REGION Network 26: pomocniczy bit ustawiania pompy dodatkowej nr1
   // Reset znacznika po udanym załączeniu pompy dodatkowej
   // Reset w wypadku braku pompy
   RUNG wire#powerrail
      I_Contact( "AlwaysTRUE" )
      wire#w1
      Contact( "Is_extras_K1_P1" )
      Contact( "IsRunNetwork_P1" )
      wire#w2
      R_Coil( #set_Motor2 )
   END_RUNG
   RUNG wire#w1
      Contact( "Is_extras_K1_P2" )
      Contact( "IsRunNetwork_P2" )
   END_RUNG wire#w2
   RUNG wire#w1
      Contact( "Is_extras_K1_P3" )
      Contact( "IsRunNetwork_P3" )
   END_RUNG wire#w2
   RUNG wire#w1
      Contact( "Is_extras_K1_P4" )
      Contact( "IsRunNetwork_P4" )
   END_RUNG wire#w2
   RUNG wire#w1
      Contact( "Reset_Motor2Alarm" )
   END_RUNG wire#w2
   RUNG wire#w1
      I_Contact( "IsModeAut" )
   END_RUNG wire#w2
   // the same network as SCL:
   IF NOT "AlwaysTRUE" AND (("Is_extras_K1_P1" AND "IsRunNetwork_P1") OR ("Is_extras_K1_P2" AND "IsRunNetwork_P2") OR ("Is_extras_K1_P3" AND "IsRunNetwork_P3") OR ("Is_extras_K1_P4" AND "IsRunNetwork_P4") OR "Reset_Motor2Alarm" OR NOT "IsModeAut") THEN
       #set_Motor2 := FALSE;
   END_IF;
END_REGION

REGION Network 27: pomocniczy bit ustawiania pompy dodatkoweo nr2
   // Reset znacznika po udanym załączeniu pompy dodatkowej
   // Reset w wypadku braku pompy
   RUNG wire#powerrail
      I_Contact( "AlwaysTRUE" )
      wire#w1
      Contact( "Is_extras_K2_P1" )
      Contact( "IsRunNetwork_P1" )
      wire#w2
      R_Coil( #set_Motor3 )
   END_RUNG
   RUNG wire#w1
      Contact( "Is_extras_K2_P2" )
      Contact( "IsRunNetwork_P2" )
   END_RUNG wire#w2
   RUNG wire#w1
      Contact( "Is_extras_K2_P3" )
      Contact( "IsRunNetwork_P3" )
   END_RUNG wire#w2
   RUNG wire#w1
      Contact( "Is_extras_K2_P4" )
      Contact( "IsRunNetwork_P4" )
   END_RUNG wire#w2
   RUNG wire#w1
      Contact( "Reset_Motor3Alarm" )
   END_RUNG wire#w2
   RUNG wire#w1
      I_Contact( "IsModeAut" )
   END_RUNG wire#w2
   // the same network as SCL:
   IF NOT "AlwaysTRUE" AND (("Is_extras_K2_P1" AND "IsRunNetwork_P1") OR ("Is_extras_K2_P2" AND "IsRunNetwork_P2") OR ("Is_extras_K2_P3" AND "IsRunNetwork_P3") OR ("Is_extras_K2_P4" AND "IsRunNetwork_P4") OR "Reset_Motor3Alarm" OR NOT "IsModeAut") THEN
       #set_Motor3 := FALSE;
   END_IF;
END_REGION

REGION Network 28: pomocniczy bit ustawiania pompy dodatkowe nr3
   // Reset znacznika po udanym załączeniu pompy dodatkowej
   // Reset w wypadku braku pompy
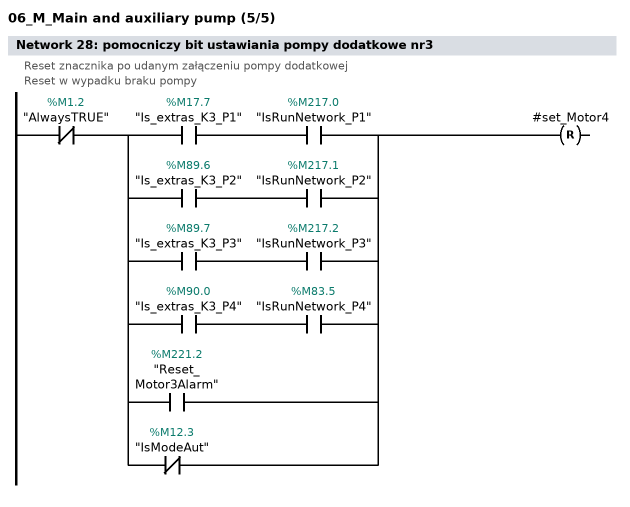
   RUNG wire#powerrail
      I_Contact( "AlwaysTRUE" )
      wire#w1
      Contact( "Is_extras_K3_P1" )
      Contact( "IsRunNetwork_P1" )
      wire#w2
      R_Coil( #set_Motor4 )
   END_RUNG
   RUNG wire#w1
      Contact( "Is_extras_K3_P2" )
      Contact( "IsRunNetwork_P2" )
   END_RUNG wire#w2
   RUNG wire#w1
      Contact( "Is_extras_K3_P3" )
      Contact( "IsRunNetwork_P3" )
   END_RUNG wire#w2
   RUNG wire#w1
      Contact( "Is_extras_K3_P4" )
      Contact( "IsRunNetwork_P4" )
   END_RUNG wire#w2
   RUNG wire#w1
      Contact( "Reset_Motor3Alarm" )
   END_RUNG wire#w2
   RUNG wire#w1
      I_Contact( "IsModeAut" )
   END_RUNG wire#w2
   // the same network as SCL:
   IF NOT "AlwaysTRUE" AND (("Is_extras_K3_P1" AND "IsRunNetwork_P1") OR ("Is_extras_K3_P2" AND "IsRunNetwork_P2") OR ("Is_extras_K3_P3" AND "IsRunNetwork_P3") OR ("Is_extras_K3_P4" AND "IsRunNetwork_P4") OR "Reset_Motor3Alarm" OR NOT "IsModeAut") THEN
       #set_Motor4 := FALSE;
   END_IF;
END_REGION
END_FUNCTION_BLOCK

FUNCTION_BLOCK "06_M_Inverter connection control"   // FB8, LAD
TITLE = Sterowanie dołączaniem styczników falownika
{ S7_Optimized_Access := 'TRUE' }
AUTHOR : rtecmer
VERSION : 0.1
// Sterowa stycznikiem pracy z falownika.
// Funkcja FB8 komutuje załaczenie stycznika FALOWNIK dla konkretnego napędu. Napędem sterowanym jest zawsze napęd przypisany do MC (czyli IsReady_MC to jest gotowość napędu sterowaniego) Na wejścia oznaczone wyróżnikiem MC podlączamy sygnały tej samej dmuchawy, której stycznikiem będziemy sterować poprzez wtjście setSUPV_FM
//  
// Sterowanie stycznikiem . Ustawianie znaczników setCMD_FM i setSUPV_FM które przekazywane są do funkcji FC3/FC1 DRV01 driver napędów. Następnie przekazywane jest do warstwy Hawtware/ OUT gdzie ustawiane jest wyjście sterownika
// stored: AutoNumber true, IsIECCheckEnabled false, IsRetainMemResEnabled false, MemoryReserve 500, SetENOAutomatically false, UDAEnableTagReadback false
   VAR_INPUT
      Is_up_Hz : Bool;
      Set_HWork_M : Bool;   // Znacznik ustawienia pracy od licznika
      setPID_Pompy : Bool;   // Znacznik załączenie, regulacji falownika
      IsRunInverter_MA : Bool;   // Potwierdzenie pracy z falownika kompresor dodatkowy 1
      IsRunNetwork_MA : Bool;   // Potwierdzenie praca z sieć dodatkowego
      IsRunInverter_MB : Bool;   // Potwierdzenie pracy z falownika kompresor dodatkowy 2
      IsRunNetwork_MB : Bool;   // Potwierdzenie praca z sieć dodatkowego
      IsRunNetwork_MC : Bool;   // Potwierdzenie pracy z sieci
      IsRunInverter_MC : Bool;   // Potwierdzenie pracy z falownika
      IsRunNetwork_MD : Bool;   // Potwierdzenie pracy z sieci
      IsRunInverter_MD : Bool;   // Potwierdzenie pracy z falownika
      FC2_Set_50H : Bool;   // Znacznik osiągnięcia czasu dla 50Hz
      IsRunInverter1 : Bool;   // Potwierdzenie pracy falownika
      AlwaysTRUE : Bool;
      IsReady_MA : Bool;   // Znacznik gotowości
      IsReady_MB : Bool;   // Znacznik gotowości
      IsReady_MC : Bool;   // Znacznik gotowości
      IsReady_MD : Bool;   // Znacznik gotowości
      IsModeAut : Bool;   // Znacznik trybu automat
      FB9_Set_Motor2 : Bool;   // Polecenie dostawienia dodatkowej nr1
      FB9_Set_Motor3 : Bool;   // Polecenie dostawienia dodatkowej nr2
      FB9_Set_Motor4 : Bool;   // Polecenie dostawienia dodatkowej nr3
      IsReady_Inverter : Bool;   // Gotowość falownika
      ResWorkInverter_to_MaxTime : Bool;   // Bit kasowania pracy falownika od maxymalnej ciągłej pracy
      number_pump : Int;   // numer pompy w instalacji
      ActivePump : Int;   // numer pompy wiodącej
   END_VAR
   VAR_OUTPUT
      setSUPV_FM : Bool;   // Znacznik polecenia startu z falownika
   END_VAR
   VAR_IN_OUT
      setCMD_FM : Bool;   // Znacznik sterowania w trybie falownik
      Timer_OFF_Inverter_M : TOF_TIME;   // Timer na blokowanie po odłączeniu stycznika falownika
      Timer_Start_Inver_M : TON_TIME;   // Timer opóźnienia załaczenia stycznika pracy z falownika
      Timer_Set50Hz_Off_Inver_M : TON_TIME;   // Timer opóźnieniawyłączeniea falownika
      Mem_Res_setCMD_MC : Bool;   // pamięć zbocza załączenia timera blokowania stycznika falowni
   END_VAR
   VAR
      IsDrive_Optimum { ExternalAccessible := 'False'; ExternalVisible := 'False'; ExternalWritable := 'False'} : Bool;   // Znacznik optymalnej ilości napędów. Jeśli False to nie przełaczaj Falowni/Sieć
      CMD_OFF_inverter { ExternalAccessible := 'False'; ExternalVisible := 'False'; ExternalWritable := 'False'} : Bool;   // Wyłączenie falownika od 50Hz i dodatkowa
      tmpOFF_inverter { ExternalAccessible := 'False'; ExternalVisible := 'False'; ExternalWritable := 'False'} : Bool;
      Network_50Hz : Bool;   // Znacznik 50 Hz podtrzymanie przełączenia na sieć
   END_VAR
   VAR_TEMP   // added for the SCL form of the ladder/FBD networks
      _w1 : Bool;
      _w2 : Bool;
   END_VAR
BEGIN

REGION Network 1: Kontrola statusu napędu
END_REGION

REGION Network 2: Histereza na dołączenie stycznika falownika
   // Sterowanie dołączeniem stycznika pracy z falownika
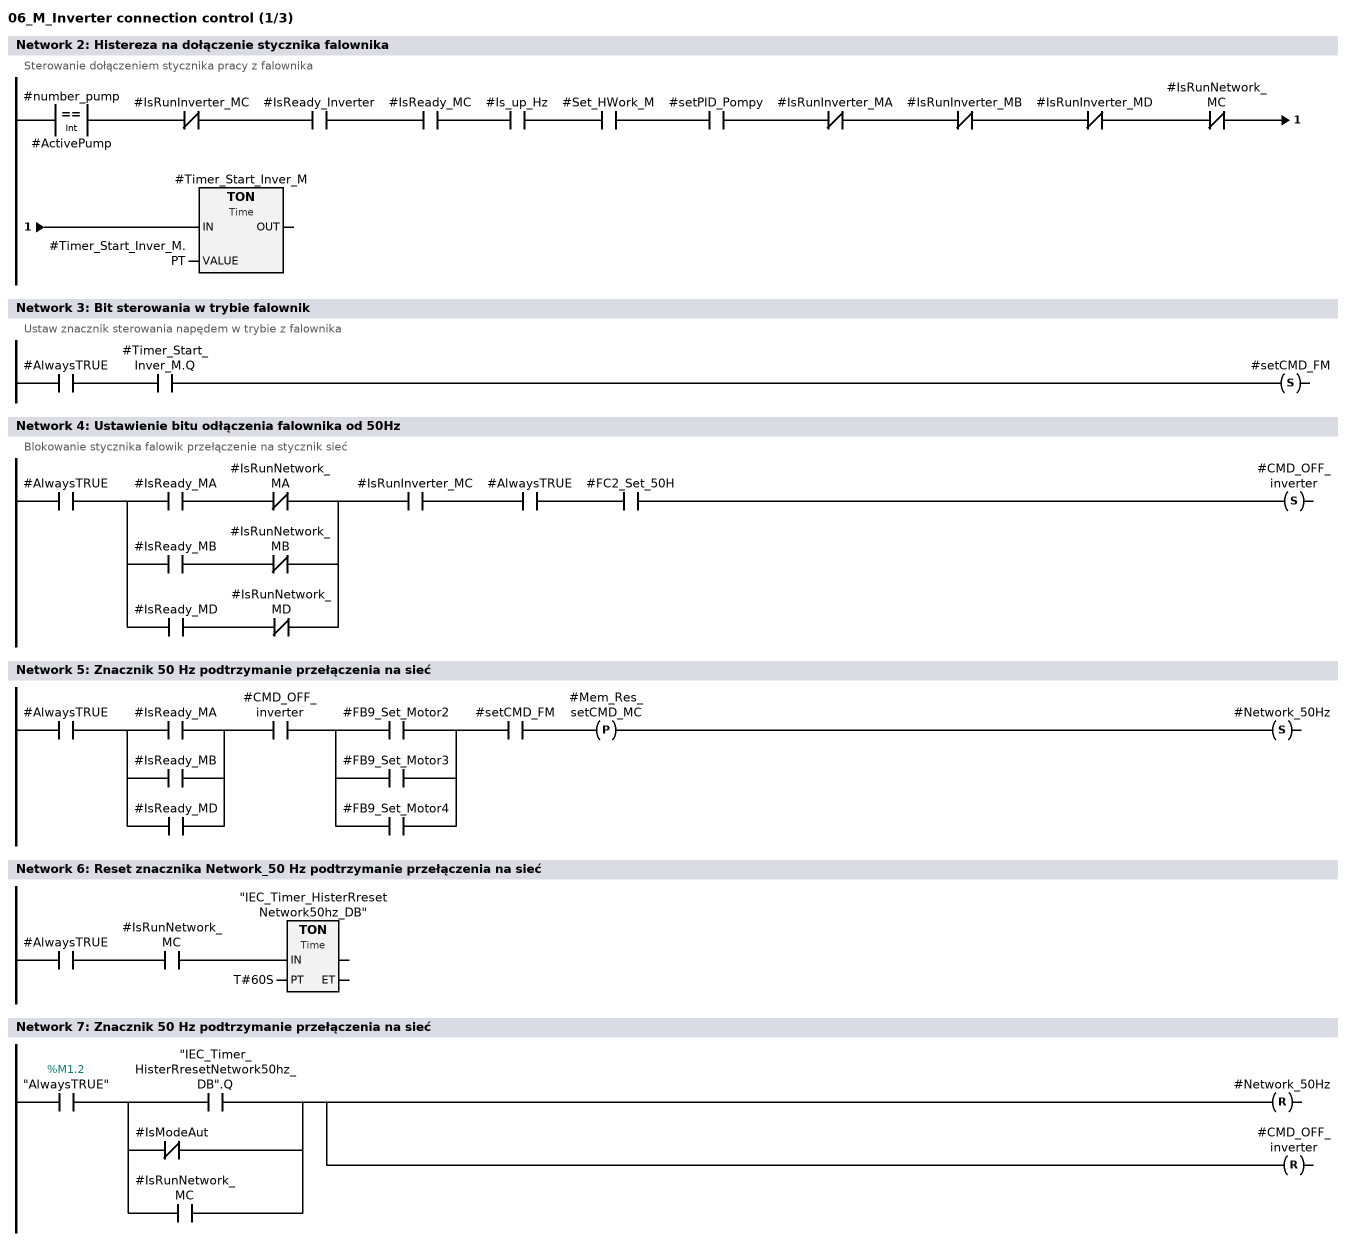
   #Timer_Start_Inver_M(IN := (#number_pump = #ActivePump) AND NOT #IsRunInverter_MC AND #IsReady_Inverter AND #IsReady_MC AND #Is_up_Hz AND #Set_HWork_M AND #setPID_Pompy AND NOT #IsRunInverter_MA AND NOT #IsRunInverter_MB AND NOT #IsRunInverter_MD AND NOT #IsRunNetwork_MC, PT := #Timer_Start_Inver_M.PT);   // TON coil
END_REGION

REGION Network 3: Bit sterowania w trybie falownik
   // Ustaw znacznik sterowania napędem w trybie z falownika
   RUNG wire#powerrail
      Contact( #AlwaysTRUE )
      Contact( #Timer_Start_Inver_M.Q )
      S_Coil( #setCMD_FM )
   END_RUNG
   // the same network as SCL:
   IF #AlwaysTRUE AND #Timer_Start_Inver_M.Q THEN #setCMD_FM := TRUE; END_IF;
END_REGION

REGION Network 4: Ustawienie bitu odłączenia falownika od 50Hz
   // Blokowanie stycznika falowik przełączenie na stycznik sieć
   RUNG wire#powerrail
      Contact( #AlwaysTRUE )
      wire#w1
      Contact( #IsReady_MA )
      I_Contact( #IsRunNetwork_MA )
      wire#w2
      Contact( #IsRunInverter_MC )
      Contact( #AlwaysTRUE )
      Contact( #FC2_Set_50H )
      S_Coil( #CMD_OFF_inverter )
   END_RUNG
   RUNG wire#w1
      Contact( #IsReady_MB )
      I_Contact( #IsRunNetwork_MB )
   END_RUNG wire#w2
   RUNG wire#w1
      Contact( #IsReady_MD )
      I_Contact( #IsRunNetwork_MD )
   END_RUNG wire#w2
   // the same network as SCL:
   IF #AlwaysTRUE AND ((#IsReady_MA AND NOT #IsRunNetwork_MA) OR (#IsReady_MB AND NOT #IsRunNetwork_MB) OR (#IsReady_MD AND NOT #IsRunNetwork_MD)) AND #IsRunInverter_MC AND #AlwaysTRUE AND #FC2_Set_50H THEN
       #CMD_OFF_inverter := TRUE;
   END_IF;
END_REGION

REGION Network 5: Znacznik 50 Hz podtrzymanie przełączenia na sieć
   RUNG wire#powerrail
      Contact( #AlwaysTRUE )
      wire#w1
      Contact( #IsReady_MA )
      wire#w2
      Contact( #CMD_OFF_inverter )
      wire#w3
      Contact( #FB9_Set_Motor2 )
      wire#w4
      Contact( #setCMD_FM )
      P_Trig( #Mem_Res_setCMD_MC )
      S_Coil( #Network_50Hz )
   END_RUNG
   RUNG wire#w1
      Contact( #IsReady_MB )
   END_RUNG wire#w2
   RUNG wire#w1
      Contact( #IsReady_MD )
   END_RUNG wire#w2
   RUNG wire#w3
      Contact( #FB9_Set_Motor3 )
   END_RUNG wire#w4
   RUNG wire#w3
      Contact( #FB9_Set_Motor4 )
   END_RUNG wire#w4
   // the same network as SCL:
   #_w1 := #AlwaysTRUE AND (#IsReady_MA OR #IsReady_MB OR #IsReady_MD) AND #CMD_OFF_inverter AND (#FB9_Set_Motor2 OR #FB9_Set_Motor3 OR #FB9_Set_Motor4) AND #setCMD_FM;
   #_w2 := #_w1 AND NOT #Mem_Res_setCMD_MC;   // rising edge
   #Mem_Res_setCMD_MC := #_w1;
   IF #_w2 THEN #Network_50Hz := TRUE; END_IF;
END_REGION

REGION Network 6: Reset znacznika Network_50 Hz podtrzymanie przełączenia na sieć
   RUNG wire#powerrail
      Contact( #AlwaysTRUE )
      Contact( #IsRunNetwork_MC )
      { S7_Templates := "time_type := Time" } "IEC_Timer_HisterRresetNetwork50hz_DB".TON(pt := T#60S, et =>)
   END_RUNG
   // the same network as SCL:
   "IEC_Timer_HisterRresetNetwork50hz_DB".TON(IN := #AlwaysTRUE AND #IsRunNetwork_MC, PT := T#60S);
END_REGION

REGION Network 7: Znacznik 50 Hz podtrzymanie przełączenia na sieć
   RUNG wire#powerrail
      Contact( "AlwaysTRUE" )
      wire#w1
      Contact( "IEC_Timer_HisterRresetNetwork50hz_DB".Q )
      wire#w2
      R_Coil( #Network_50Hz )
   END_RUNG
   RUNG wire#w1
      I_Contact( #IsModeAut )
   END_RUNG wire#w2
   RUNG wire#w1
      Contact( #IsRunNetwork_MC )
   END_RUNG wire#w2
   RUNG wire#w2
      R_Coil( #CMD_OFF_inverter )
   END_RUNG
   // the same network as SCL:
   IF "AlwaysTRUE" AND ("IEC_Timer_HisterRresetNetwork50hz_DB".Q OR NOT #IsModeAut OR #IsRunNetwork_MC) THEN
       #Network_50Hz := FALSE;
       #CMD_OFF_inverter := FALSE;
   END_IF;
END_REGION

REGION Network 8: Timer blokowania po odłączenieu stycznika falownik
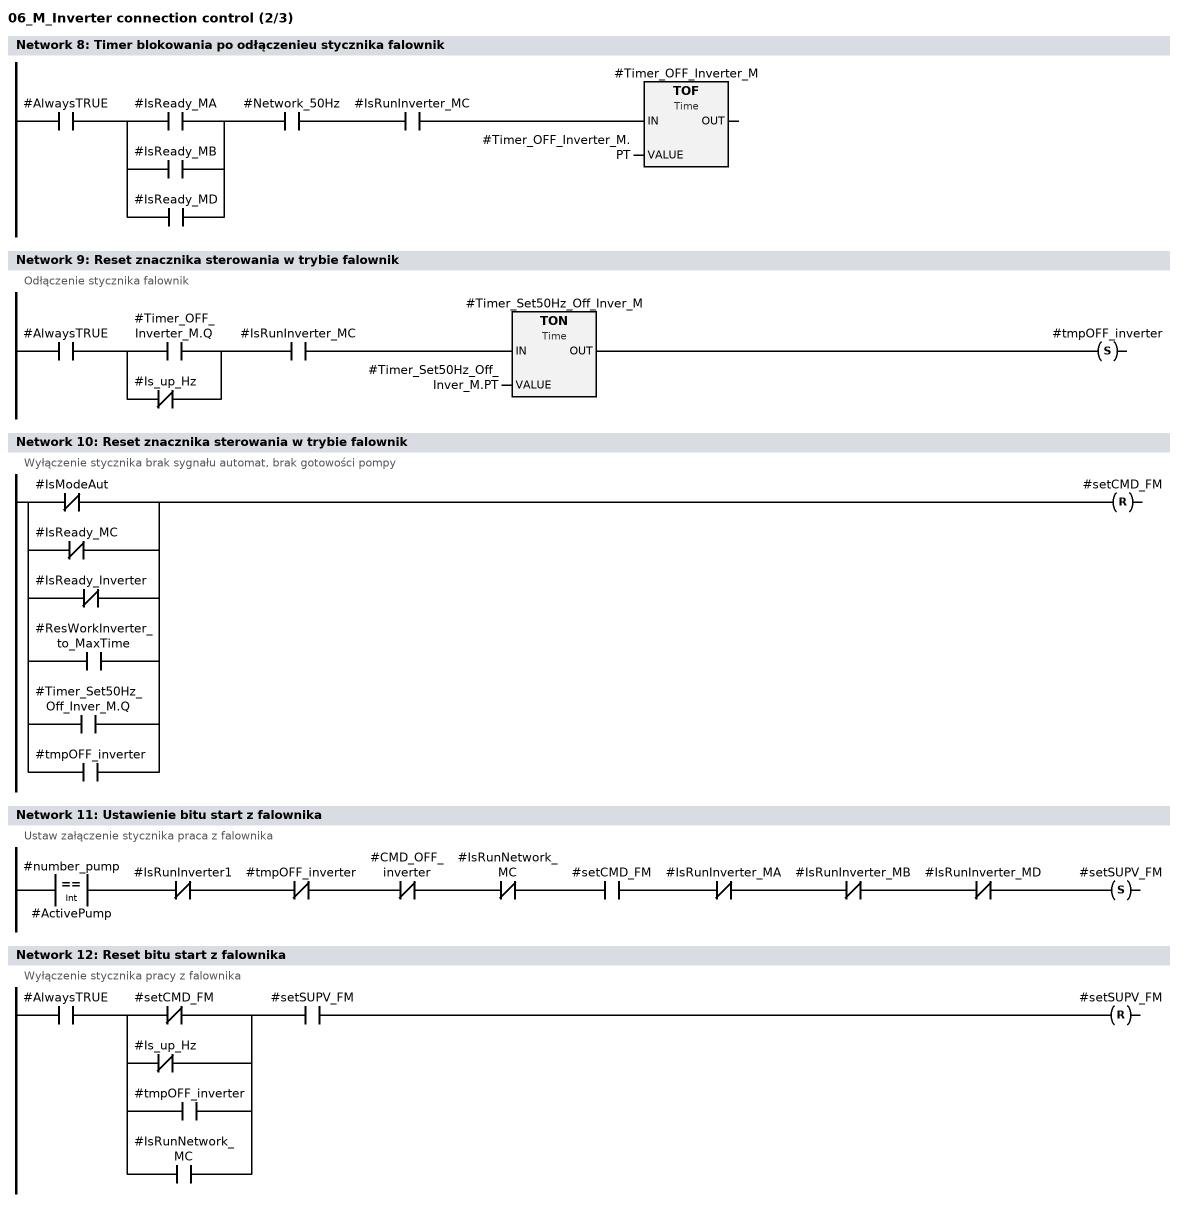
   #Timer_OFF_Inverter_M(IN := #AlwaysTRUE AND (#IsReady_MA OR #IsReady_MB OR #IsReady_MD) AND #Network_50Hz AND #IsRunInverter_MC, PT := #Timer_OFF_Inverter_M.PT);   // TOF coil
END_REGION

REGION Network 9: Reset znacznika sterowania w trybie falownik
   // Odłączenie stycznika falownik
   #_w1 := #AlwaysTRUE AND (#Timer_OFF_Inverter_M.Q OR NOT #Is_up_Hz) AND #IsRunInverter_MC;
   #Timer_Set50Hz_Off_Inver_M(IN := #_w1, PT := #Timer_Set50Hz_Off_Inver_M.PT);   // TON coil
   IF #_w1 THEN #tmpOFF_inverter := TRUE; END_IF;
END_REGION

REGION Network 10: Reset znacznika sterowania w trybie falownik
   // Wyłączenie stycznika brak sygnału automat, brak gotowości pompy
   RUNG wire#powerrail
      I_Contact( #IsModeAut )
      wire#w1
      R_Coil( #setCMD_FM )
   END_RUNG
   RUNG wire#powerrail
      I_Contact( #IsReady_MC )
   END_RUNG wire#w1
   RUNG wire#powerrail
      I_Contact( #IsReady_Inverter )
   END_RUNG wire#w1
   RUNG wire#powerrail
      Contact( #ResWorkInverter_to_MaxTime )
   END_RUNG wire#w1
   RUNG wire#powerrail
      Contact( #Timer_Set50Hz_Off_Inver_M.Q )
   END_RUNG wire#w1
   RUNG wire#powerrail
      Contact( #tmpOFF_inverter )
   END_RUNG wire#w1
   // the same network as SCL:
   IF NOT #IsModeAut OR NOT #IsReady_MC OR NOT #IsReady_Inverter OR #ResWorkInverter_to_MaxTime OR #Timer_Set50Hz_Off_Inver_M.Q OR #tmpOFF_inverter THEN
       #setCMD_FM := FALSE;
   END_IF;
END_REGION

REGION Network 11: Ustawienie bitu start z falownika
   // Ustaw załączenie stycznika praca z falownika
   RUNG wire#powerrail
      { S7_Templates := "SrcType := Int" } EQ_Contact(in1 := #number_pump, in2 := #ActivePump)
      I_Contact( #IsRunInverter1 )
      I_Contact( #tmpOFF_inverter )
      I_Contact( #CMD_OFF_inverter )
      I_Contact( #IsRunNetwork_MC )
      Contact( #setCMD_FM )
      I_Contact( #IsRunInverter_MA )
      I_Contact( #IsRunInverter_MB )
      I_Contact( #IsRunInverter_MD )
      S_Coil( #setSUPV_FM )
   END_RUNG
   // the same network as SCL:
   IF (#number_pump = #ActivePump) AND NOT #IsRunInverter1 AND NOT #tmpOFF_inverter AND NOT #CMD_OFF_inverter AND NOT #IsRunNetwork_MC AND #setCMD_FM AND NOT #IsRunInverter_MA AND NOT #IsRunInverter_MB AND NOT #IsRunInverter_MD THEN
       #setSUPV_FM := TRUE;
   END_IF;
END_REGION

REGION Network 12: Reset bitu start z falownika
   // Wyłączenie stycznika pracy z falownika
   RUNG wire#powerrail
      Contact( #AlwaysTRUE )
      wire#w1
      I_Contact( #setCMD_FM )
      wire#w2
      Contact( #setSUPV_FM )
      R_Coil( #setSUPV_FM )
   END_RUNG
   RUNG wire#w1
      I_Contact( #Is_up_Hz )
   END_RUNG wire#w2
   RUNG wire#w1
      Contact( #tmpOFF_inverter )
   END_RUNG wire#w2
   RUNG wire#w1
      Contact( #IsRunNetwork_MC )
   END_RUNG wire#w2
   // the same network as SCL:
   IF #AlwaysTRUE AND (NOT #setCMD_FM OR NOT #Is_up_Hz OR #tmpOFF_inverter OR #IsRunNetwork_MC) AND #setSUPV_FM THEN
       #setSUPV_FM := FALSE;
   END_IF;
END_REGION

REGION Network 13: Znacznik polecenia stop z falownika
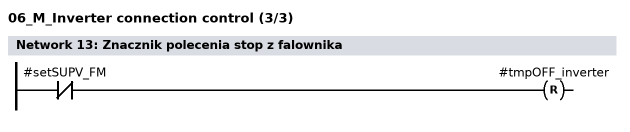
   RUNG wire#powerrail
      I_Contact( #setSUPV_FM )
      R_Coil( #tmpOFF_inverter )
   END_RUNG
   // the same network as SCL:
   IF NOT #setSUPV_FM THEN #tmpOFF_inverter := FALSE; END_IF;
END_REGION
END_FUNCTION_BLOCK

FUNCTION "06_M_Working Mode Correction" : Void   // FC34, LAD
TITLE = potrzymanie trybu
{ S7_Optimized_Access := 'TRUE' }
AUTHOR : rtecmer
VERSION : 0.1
// z powodu P1 dodanyblok potzymujący tryb pracy napędów podczas przełączania falowni / siec
// stored: AutoNumber true, IsIECCheckEnabled false, SetENOAutomatically false, UDAEnableTagReadback false
   VAR_TEMP   // added for the SCL form of the ladder/FBD networks
      _w1 : Bool;
   END_VAR
BEGIN

REGION Network 2: Ustawienie pracy [Automat]
   // Ustawienie bitu [Automat] przełacznikiem trybu pracy
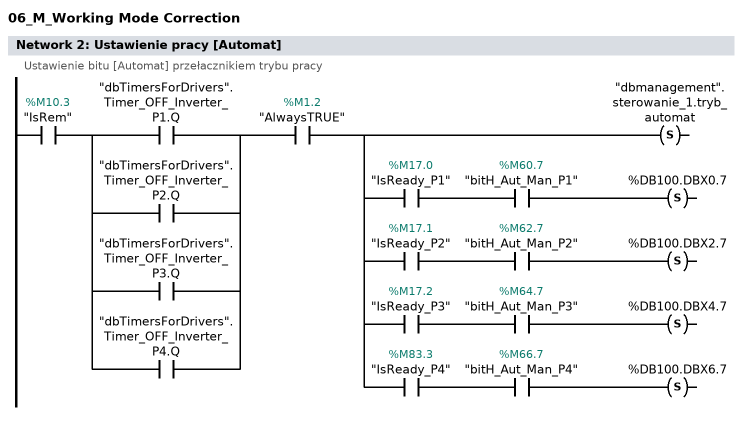
   RUNG wire#powerrail
      Contact( "IsRem" )
      wire#w1
      Contact( "dbTimersForDrivers".Timer_OFF_Inverter_P1.Q )
      wire#w2
      Contact( "AlwaysTRUE" )
      wire#w3
      S_Coil( "dbmanagement".sterowanie_1.tryb_automat )
   END_RUNG
   RUNG wire#w1
      Contact( "dbTimersForDrivers".Timer_OFF_Inverter_P2.Q )
   END_RUNG wire#w2
   RUNG wire#w1
      Contact( "dbTimersForDrivers".Timer_OFF_Inverter_P3.Q )
   END_RUNG wire#w2
   RUNG wire#w1
      Contact( "dbTimersForDrivers".Timer_OFF_Inverter_P4.Q )
   END_RUNG wire#w2
   RUNG wire#w3
      Contact( "IsReady_P1" )
      Contact( "bitH_Aut_Man_P1" )
      S_Coil( %DB100.DBX0.7 )
   END_RUNG
   RUNG wire#w3
      Contact( "IsReady_P2" )
      Contact( "bitH_Aut_Man_P2" )
      S_Coil( %DB100.DBX2.7 )
   END_RUNG
   RUNG wire#w3
      Contact( "IsReady_P3" )
      Contact( "bitH_Aut_Man_P3" )
      S_Coil( %DB100.DBX4.7 )
   END_RUNG
   RUNG wire#w3
      Contact( "IsReady_P4" )
      Contact( "bitH_Aut_Man_P4" )
      S_Coil( %DB100.DBX6.7 )
   END_RUNG
   // the same network as SCL:
   #_w1 := "IsRem" AND ("dbTimersForDrivers".Timer_OFF_Inverter_P1.Q OR "dbTimersForDrivers".Timer_OFF_Inverter_P2.Q OR "dbTimersForDrivers".Timer_OFF_Inverter_P3.Q OR "dbTimersForDrivers".Timer_OFF_Inverter_P4.Q) AND "AlwaysTRUE";
   IF #_w1 THEN "dbmanagement".sterowanie_1.tryb_automat := TRUE; END_IF;
   IF #_w1 AND "IsReady_P1" AND "bitH_Aut_Man_P1" THEN %DB100.DBX0.7 := TRUE; END_IF;
   IF #_w1 AND "IsReady_P2" AND "bitH_Aut_Man_P2" THEN %DB100.DBX2.7 := TRUE; END_IF;
   IF #_w1 AND "IsReady_P3" AND "bitH_Aut_Man_P3" THEN %DB100.DBX4.7 := TRUE; END_IF;
   IF #_w1 AND "IsReady_P4" AND "bitH_Aut_Man_P4" THEN %DB100.DBX6.7 := TRUE; END_IF;
END_REGION
END_FUNCTION

FUNCTION_BLOCK "06_M_Inverte control"   // FB11, LAD
TITLE = Control of Inverters
{ S7_Optimized_Access := 'TRUE' }
AUTHOR : rtecmer
VERSION : 0.1
// Sterowanie przekaćnikiem załączającym falownik do pracy
// stored: AutoNumber true, IsIECCheckEnabled false, IsRetainMemResEnabled false, MemoryReserve 500, SetENOAutomatically false, UDAEnableTagReadback false
   VAR_INPUT
      IsModeAut : Bool;   // Znacznik tryb automat dla pomp
      AlwaysTRUE : Bool;
      Set_HWork_P1 : Bool;   // Znacznik ustawienia pracy od licznika pracy
      Set_HWork_P2 : Bool;   // Znacznik ustawienia pracy od licznika pracy
      Set_HWork_P3 : Bool;   // Znacznik ustawienia pracy od licznika pracy
      Set_HWork_P4 : Bool;
      setPID_Pomp : Bool;   // Znacznik załączenie, regulacji falownika
      Is_loading_K3 : Bool;   // Znacznik pompy wiodącej
      IsRunInverter_P4 : Bool;
      IsRunInverter_P3 : Bool;   // Potwierdzenie załączenie stycznika falownik pompy
      IsRunInverter_P2 : Bool;   // Potwierdzenie załączenie stycznika falownik pompy
      IsRunInverter_P1 : Bool;   // Potwierdzenie załączenie stycznika falownik pompy
      Bit_Aut_P1 : Bool;   // Bit tryb prac automat
      Bit_Aut_P2 : Bool;   // Bit tryb prac automat
      Bit_Aut_P3 : Bool;   // Bit tryb prac automat
      Bit_Aut_P4 : Bool;
      IsRunNetwork_P1 : Bool;   // Potwierdzenie załączenie stycznika sieć
      IsRunNetwork_P2 : Bool := false;   // Potwierdzenie załączenie stycznika sieć
      IsRunNetwork_P3 : Bool := false;   // Potwierdzenie załączenie stycznika sieć
      IsRunNetwork_P4 : Bool;
   END_VAR
   VAR_OUTPUT
      CMD_start_stop_inverter : Bool;   // Przekaźnik sterowania załączaniem falownika
   END_VAR
   VAR
      Res_upHz : Bool;   // Reset znacznika up_Hz wyłaczenie dodatkowe
   END_VAR
BEGIN

REGION Network 1: Reset bitu pomocniczego ustalenia przyrostu Hz
   // Kasowanie podczas rozruchu po restarcie
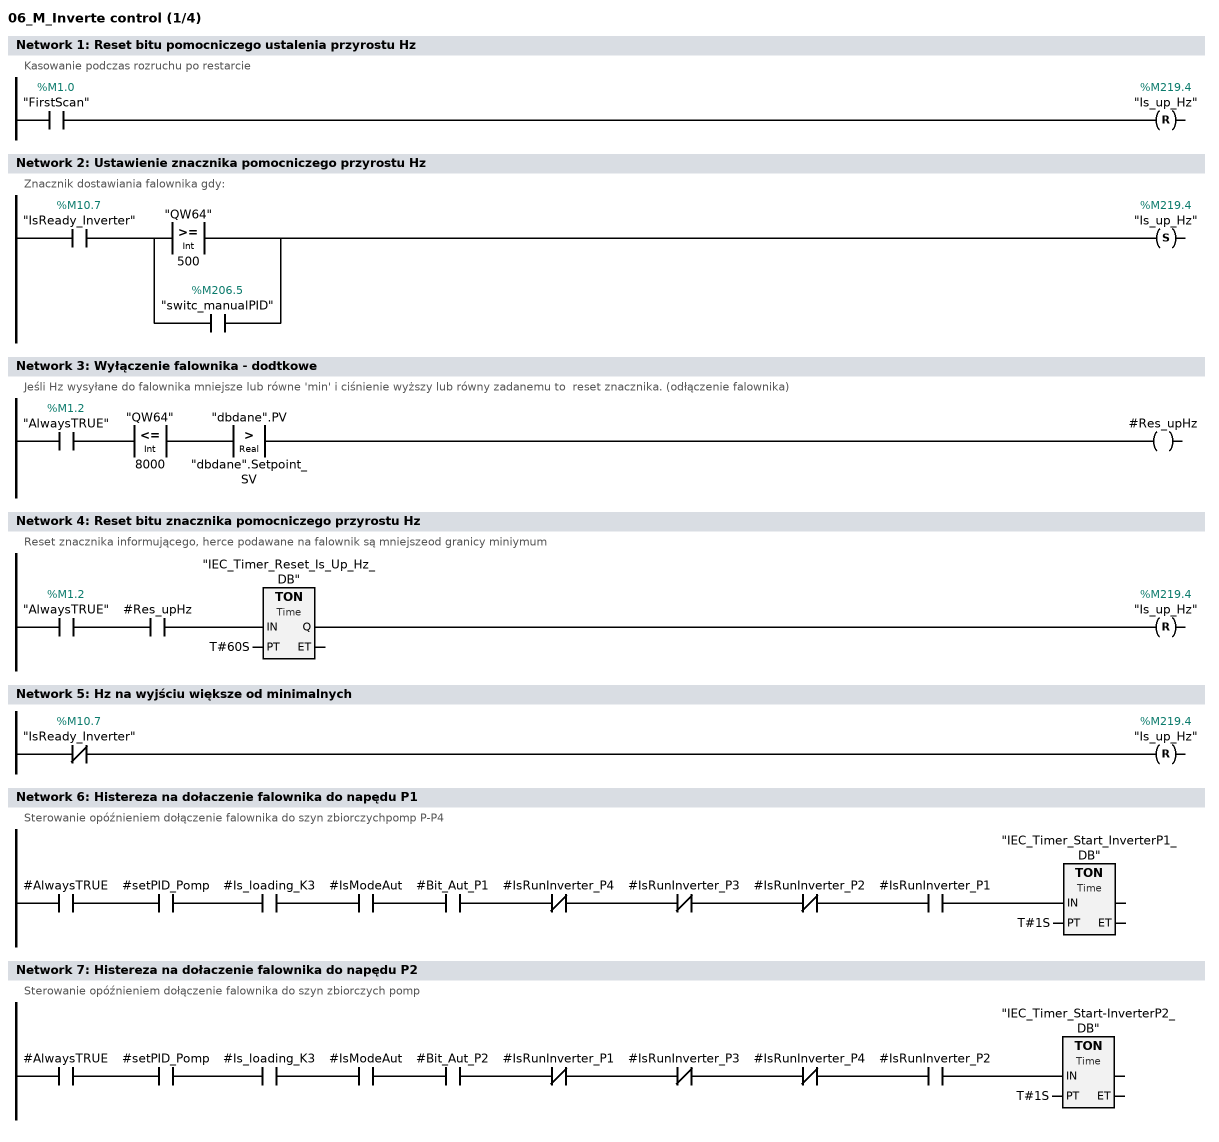
   RUNG wire#powerrail
      Contact( "FirstScan" )
      R_Coil( "Is_up_Hz" )
   END_RUNG
   // the same network as SCL:
   IF "FirstScan" THEN "Is_up_Hz" := FALSE; END_IF;
END_REGION

REGION Network 2: Ustawienie znacznika pomocniczego przyrostu Hz
   // Znacznik dostawiania falownika gdy:
   RUNG wire#powerrail
      Contact( "IsReady_Inverter" )
      wire#w1
      { S7_Templates := "SrcType := Int" } GE_Contact(in1 := "QW64", in2 := 500)
      wire#w2
      S_Coil( "Is_up_Hz" )
   END_RUNG
   RUNG wire#w1
      Contact( "switc_manualPID" )
   END_RUNG wire#w2
   // the same network as SCL:
   IF "IsReady_Inverter" AND (("QW64" >= 500) OR "switc_manualPID") THEN "Is_up_Hz" := TRUE; END_IF;
END_REGION

REGION Network 3: Wyłączenie falownika - dodtkowe
   // Jeśli Hz wysyłane do falownika mniejsze lub równe 'min' i ciśnienie wyższy lub równy zadanemu to  reset znacznika. (odłączenie falownika)
   RUNG wire#powerrail
      Contact( "AlwaysTRUE" )
      { S7_Templates := "SrcType := Int" } LE_Contact(in1 := "QW64", in2 := 8000)
      { S7_Templates := "SrcType := Real" } GT_Contact(in1 := "dbdane".PV, in2 := "dbdane".Setpoint_SV)
      Coil( #Res_upHz )
   END_RUNG
   // the same network as SCL:
   #Res_upHz := "AlwaysTRUE" AND ("QW64" <= 8000) AND ("dbdane".PV > "dbdane".Setpoint_SV);
END_REGION

REGION Network 4: Reset bitu znacznika pomocniczego przyrostu Hz
   // Reset znacznika informującego, herce podawane na falownik są mniejszeod granicy miniymum
   RUNG wire#powerrail
      Contact( "AlwaysTRUE" )
      Contact( #Res_upHz )
      { S7_Templates := "time_type := Time" } "IEC_Timer_Reset_Is_Up_Hz_DB".TON(pt := T#60S, et =>)
      R_Coil( "Is_up_Hz" )
   END_RUNG
   // the same network as SCL:
   "IEC_Timer_Reset_Is_Up_Hz_DB".TON(IN := "AlwaysTRUE" AND #Res_upHz, PT := T#60S);
   IF "IEC_Timer_Reset_Is_Up_Hz_DB".Q THEN "Is_up_Hz" := FALSE; END_IF;
END_REGION

REGION Network 5: Hz na wyjściu większe od minimalnych
   RUNG wire#powerrail
      I_Contact( "IsReady_Inverter" )
      R_Coil( "Is_up_Hz" )
   END_RUNG
   // the same network as SCL:
   IF NOT "IsReady_Inverter" THEN "Is_up_Hz" := FALSE; END_IF;
END_REGION

REGION Network 6: Histereza na dołaczenie falownika do napędu P1
   // Sterowanie opóźnieniem dołączenie falownika do szyn zbiorczychpomp P-P4
   RUNG wire#powerrail
      Contact( #AlwaysTRUE )
      Contact( #setPID_Pomp )
      Contact( #Is_loading_K3 )
      Contact( #IsModeAut )
      Contact( #Bit_Aut_P1 )
      I_Contact( #IsRunInverter_P4 )
      I_Contact( #IsRunInverter_P3 )
      I_Contact( #IsRunInverter_P2 )
      Contact( #IsRunInverter_P1 )
      { S7_Templates := "time_type := Time" } "IEC_Timer_Start_InverterP1_DB".TON(pt := T#1S, et =>)
   END_RUNG
   // the same network as SCL:
   "IEC_Timer_Start_InverterP1_DB".TON(IN := #AlwaysTRUE AND #setPID_Pomp AND #Is_loading_K3 AND #IsModeAut AND #Bit_Aut_P1 AND NOT #IsRunInverter_P4 AND NOT #IsRunInverter_P3 AND NOT #IsRunInverter_P2 AND #IsRunInverter_P1,
                           PT := T#1S);
END_REGION

REGION Network 7: Histereza na dołaczenie falownika do napędu P2
   // Sterowanie opóźnieniem dołączenie falownika do szyn zbiorczych pomp
   RUNG wire#powerrail
      Contact( #AlwaysTRUE )
      Contact( #setPID_Pomp )
      Contact( #Is_loading_K3 )
      Contact( #IsModeAut )
      Contact( #Bit_Aut_P2 )
      I_Contact( #IsRunInverter_P1 )
      I_Contact( #IsRunInverter_P3 )
      I_Contact( #IsRunInverter_P4 )
      Contact( #IsRunInverter_P2 )
      { S7_Templates := "time_type := Time" } "IEC_Timer_Start-InverterP2_DB".TON(pt := T#1S, et =>)
   END_RUNG
   // the same network as SCL:
   "IEC_Timer_Start-InverterP2_DB".TON(IN := #AlwaysTRUE AND #setPID_Pomp AND #Is_loading_K3 AND #IsModeAut AND #Bit_Aut_P2 AND NOT #IsRunInverter_P1 AND NOT #IsRunInverter_P3 AND NOT #IsRunInverter_P4 AND #IsRunInverter_P2,
                           PT := T#1S);
END_REGION

REGION Network 8: Histereza na dołaczenie falownika do napędu P3
   // Sterowanie opóźnieniem dołączenie falownika do szyn zbiorczych kompresorów
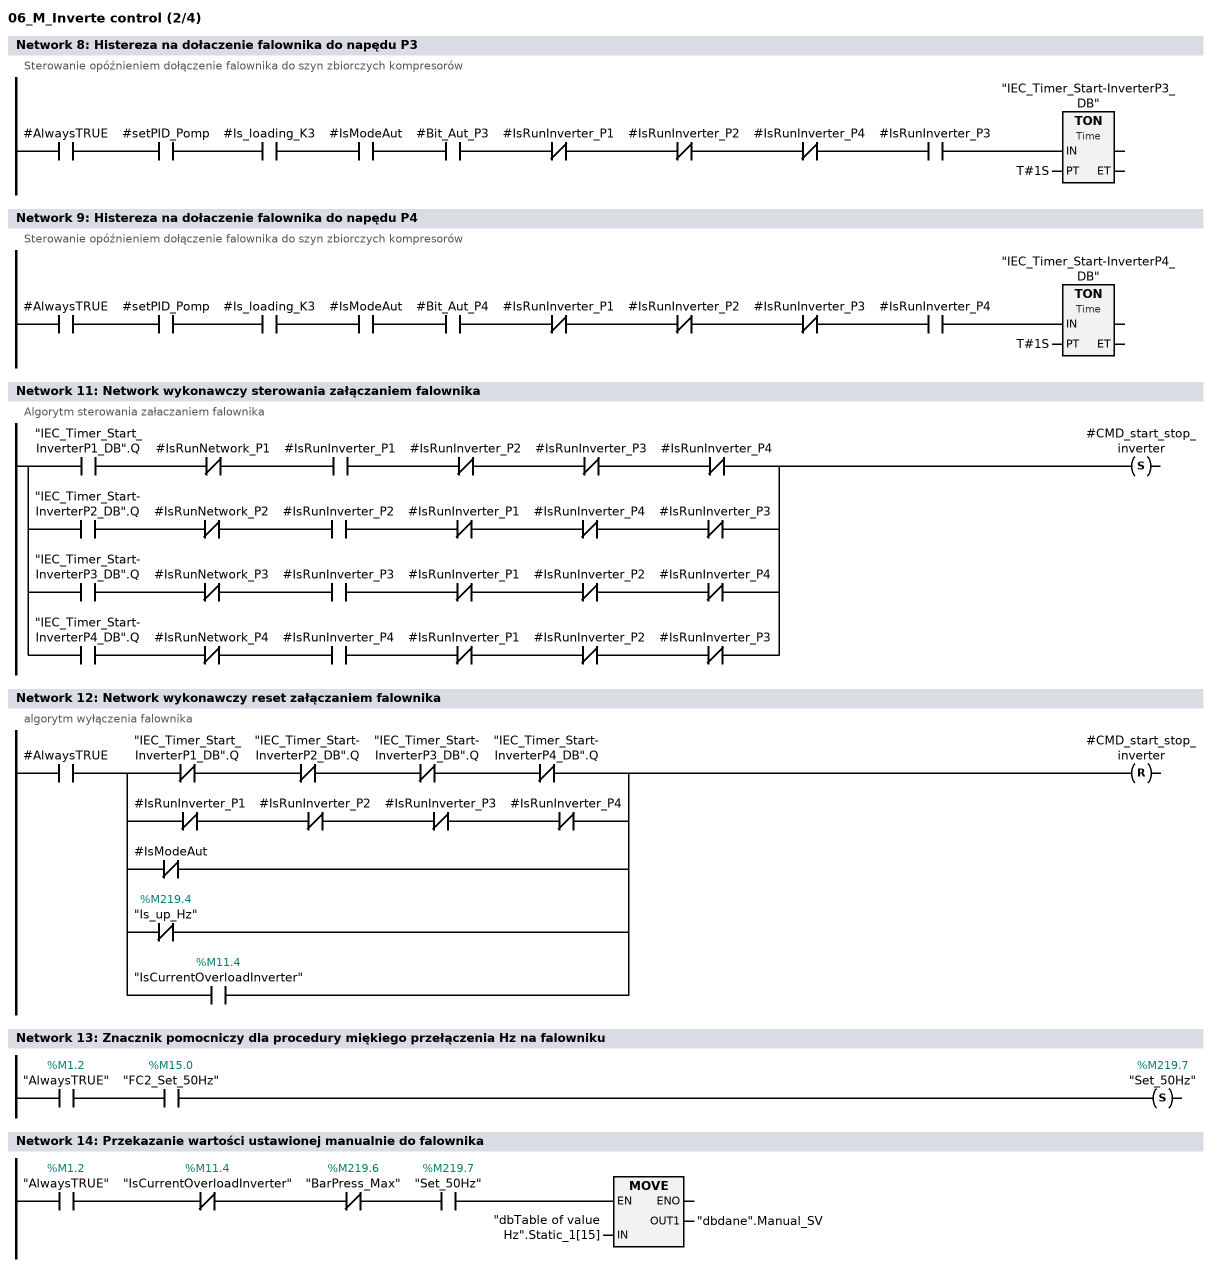
   RUNG wire#powerrail
      Contact( #AlwaysTRUE )
      Contact( #setPID_Pomp )
      Contact( #Is_loading_K3 )
      Contact( #IsModeAut )
      Contact( #Bit_Aut_P3 )
      I_Contact( #IsRunInverter_P1 )
      I_Contact( #IsRunInverter_P2 )
      I_Contact( #IsRunInverter_P4 )
      Contact( #IsRunInverter_P3 )
      { S7_Templates := "time_type := Time" } "IEC_Timer_Start-InverterP3_DB".TON(pt := T#1S, et =>)
   END_RUNG
   // the same network as SCL:
   "IEC_Timer_Start-InverterP3_DB".TON(IN := #AlwaysTRUE AND #setPID_Pomp AND #Is_loading_K3 AND #IsModeAut AND #Bit_Aut_P3 AND NOT #IsRunInverter_P1 AND NOT #IsRunInverter_P2 AND NOT #IsRunInverter_P4 AND #IsRunInverter_P3,
                           PT := T#1S);
END_REGION

REGION Network 9: Histereza na dołaczenie falownika do napędu P4
   // Sterowanie opóźnieniem dołączenie falownika do szyn zbiorczych kompresorów
   RUNG wire#powerrail
      Contact( #AlwaysTRUE )
      Contact( #setPID_Pomp )
      Contact( #Is_loading_K3 )
      Contact( #IsModeAut )
      Contact( #Bit_Aut_P4 )
      I_Contact( #IsRunInverter_P1 )
      I_Contact( #IsRunInverter_P2 )
      I_Contact( #IsRunInverter_P3 )
      Contact( #IsRunInverter_P4 )
      { S7_Templates := "time_type := Time" } "IEC_Timer_Start-InverterP4_DB".TON(pt := T#1S, et =>)
   END_RUNG
   // the same network as SCL:
   "IEC_Timer_Start-InverterP4_DB".TON(IN := #AlwaysTRUE AND #setPID_Pomp AND #Is_loading_K3 AND #IsModeAut AND #Bit_Aut_P4 AND NOT #IsRunInverter_P1 AND NOT #IsRunInverter_P2 AND NOT #IsRunInverter_P3 AND #IsRunInverter_P4,
                           PT := T#1S);
END_REGION

REGION Network 11: Network wykonawczy sterowania załączaniem falownika
   // Algorytm sterowania załaczaniem falownika
   RUNG wire#powerrail
      Contact( "IEC_Timer_Start_InverterP1_DB".Q )
      I_Contact( #IsRunNetwork_P1 )
      Contact( #IsRunInverter_P1 )
      I_Contact( #IsRunInverter_P2 )
      I_Contact( #IsRunInverter_P3 )
      I_Contact( #IsRunInverter_P4 )
      wire#w1
      S_Coil( #CMD_start_stop_inverter )
   END_RUNG
   RUNG wire#powerrail
      Contact( "IEC_Timer_Start-InverterP2_DB".Q )
      I_Contact( #IsRunNetwork_P2 )
      Contact( #IsRunInverter_P2 )
      I_Contact( #IsRunInverter_P1 )
      I_Contact( #IsRunInverter_P4 )
      I_Contact( #IsRunInverter_P3 )
   END_RUNG wire#w1
   RUNG wire#powerrail
      Contact( "IEC_Timer_Start-InverterP3_DB".Q )
      I_Contact( #IsRunNetwork_P3 )
      Contact( #IsRunInverter_P3 )
      I_Contact( #IsRunInverter_P1 )
      I_Contact( #IsRunInverter_P2 )
      I_Contact( #IsRunInverter_P4 )
   END_RUNG wire#w1
   RUNG wire#powerrail
      Contact( "IEC_Timer_Start-InverterP4_DB".Q )
      I_Contact( #IsRunNetwork_P4 )
      Contact( #IsRunInverter_P4 )
      I_Contact( #IsRunInverter_P1 )
      I_Contact( #IsRunInverter_P2 )
      I_Contact( #IsRunInverter_P3 )
   END_RUNG wire#w1
   // the same network as SCL:
   IF ("IEC_Timer_Start_InverterP1_DB".Q AND NOT #IsRunNetwork_P1 AND #IsRunInverter_P1 AND NOT #IsRunInverter_P2 AND NOT #IsRunInverter_P3 AND NOT #IsRunInverter_P4) OR ("IEC_Timer_Start-InverterP2_DB".Q AND NOT #IsRunNetwork_P2 AND #IsRunInverter_P2 AND NOT #IsRunInverter_P1 AND NOT #IsRunInverter_P4 AND NOT #IsRunInverter_P3) OR ("IEC_Timer_Start-InverterP3_DB".Q AND NOT #IsRunNetwork_P3 AND #IsRunInverter_P3 AND NOT #IsRunInverter_P1 AND NOT #IsRunInverter_P2 AND NOT #IsRunInverter_P4) OR ("IEC_Timer_Start-InverterP4_DB".Q AND NOT #IsRunNetwork_P4 AND #IsRunInverter_P4 AND NOT #IsRunInverter_P1 AND NOT #IsRunInverter_P2 AND NOT #IsRunInverter_P3) THEN
       #CMD_start_stop_inverter := TRUE;
   END_IF;
END_REGION

REGION Network 12: Network wykonawczy reset załączaniem falownika
   // algorytm wyłączenia falownika
   RUNG wire#powerrail
      Contact( #AlwaysTRUE )
      wire#w1
      I_Contact( "IEC_Timer_Start_InverterP1_DB".Q )
      I_Contact( "IEC_Timer_Start-InverterP2_DB".Q )
      I_Contact( "IEC_Timer_Start-InverterP3_DB".Q )
      I_Contact( "IEC_Timer_Start-InverterP4_DB".Q )
      wire#w2
      R_Coil( #CMD_start_stop_inverter )
   END_RUNG
   RUNG wire#w1
      I_Contact( #IsRunInverter_P1 )
      I_Contact( #IsRunInverter_P2 )
      I_Contact( #IsRunInverter_P3 )
      I_Contact( #IsRunInverter_P4 )
   END_RUNG wire#w2
   RUNG wire#w1
      I_Contact( #IsModeAut )
   END_RUNG wire#w2
   RUNG wire#w1
      I_Contact( "Is_up_Hz" )
   END_RUNG wire#w2
   RUNG wire#w1
      Contact( "IsCurrentOverloadInverter" )
   END_RUNG wire#w2
   // the same network as SCL:
   IF #AlwaysTRUE AND ((NOT "IEC_Timer_Start_InverterP1_DB".Q AND NOT "IEC_Timer_Start-InverterP2_DB".Q AND NOT "IEC_Timer_Start-InverterP3_DB".Q AND NOT "IEC_Timer_Start-InverterP4_DB".Q) OR (NOT #IsRunInverter_P1 AND NOT #IsRunInverter_P2 AND NOT #IsRunInverter_P3 AND NOT #IsRunInverter_P4) OR NOT #IsModeAut OR NOT "Is_up_Hz" OR "IsCurrentOverloadInverter") THEN
       #CMD_start_stop_inverter := FALSE;
   END_IF;
END_REGION

REGION Network 13: Znacznik pomocniczy dla procedury miękiego przełączenia Hz na falowniku
   RUNG wire#powerrail
      Contact( "AlwaysTRUE" )
      Contact( "FC2_Set_50Hz" )
      S_Coil( "Set_50Hz" )
   END_RUNG
   // the same network as SCL:
   IF "AlwaysTRUE" AND "FC2_Set_50Hz" THEN "Set_50Hz" := TRUE; END_IF;
END_REGION

REGION Network 14: Przekazanie wartości ustawionej manualnie do falownika
   RUNG wire#powerrail
      Contact( "AlwaysTRUE" )
      I_Contact( "IsCurrentOverloadInverter" )
      I_Contact( "BarPress_Max" )
      Contact( "Set_50Hz" )
      Move(in := "dbTable of value Hz".Static_1[15], out1 => "dbdane".Manual_SV)
   END_RUNG
   // the same network as SCL:
   IF "AlwaysTRUE" AND NOT "IsCurrentOverloadInverter" AND NOT "BarPress_Max" AND "Set_50Hz" THEN
       "dbdane".Manual_SV := "dbTable of value Hz".Static_1[15];
   END_IF;
END_REGION

REGION Network 15: Przekazanie wartości ustawionej manualnie do falownika gdy awaria max ciśnienie
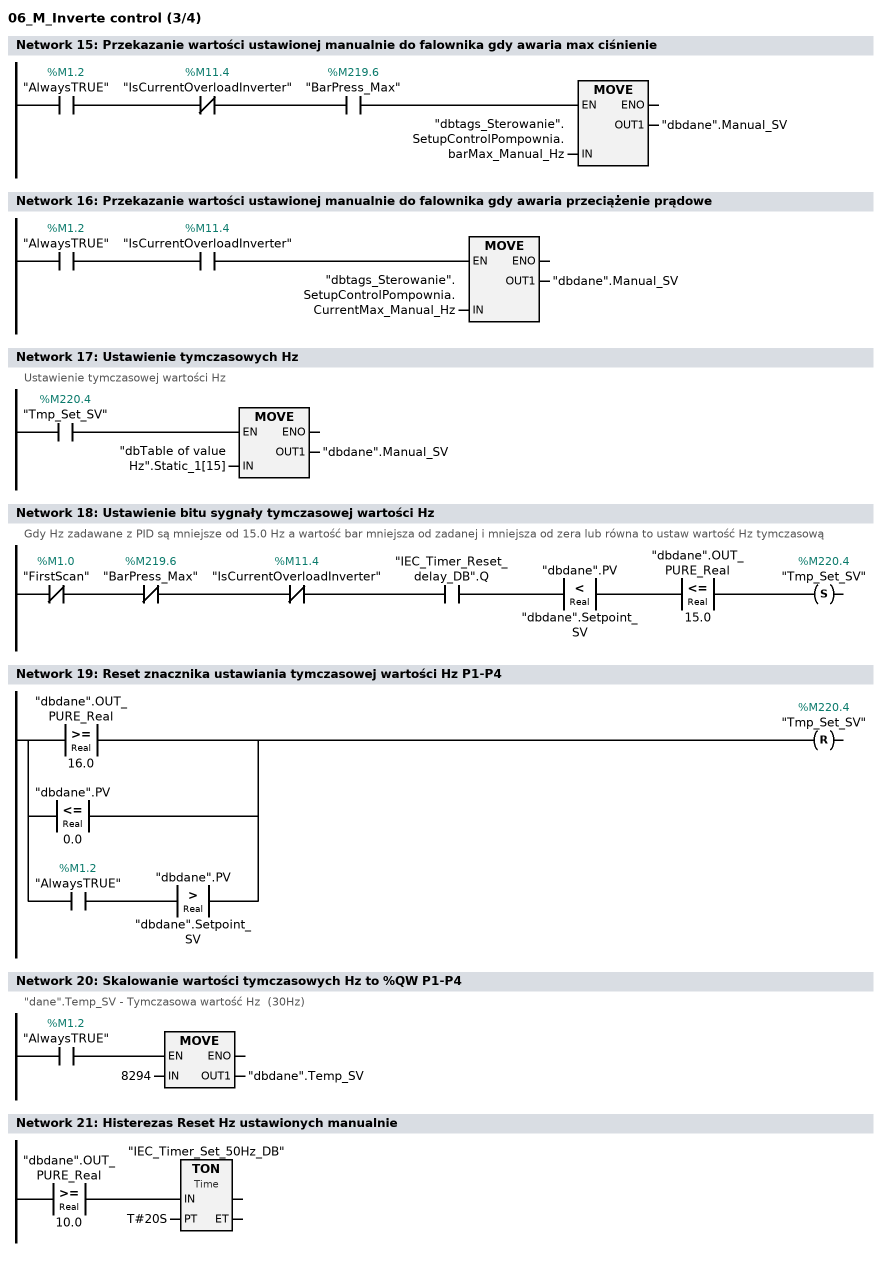
   RUNG wire#powerrail
      Contact( "AlwaysTRUE" )
      I_Contact( "IsCurrentOverloadInverter" )
      Contact( "BarPress_Max" )
      Move(in := "dbtags_Sterowanie".SetupControlPompownia.barMax_Manual_Hz, out1 => "dbdane".Manual_SV)
   END_RUNG
   // the same network as SCL:
   IF "AlwaysTRUE" AND NOT "IsCurrentOverloadInverter" AND "BarPress_Max" THEN
       "dbdane".Manual_SV := "dbtags_Sterowanie".SetupControlPompownia.barMax_Manual_Hz;
   END_IF;
END_REGION

REGION Network 16: Przekazanie wartości ustawionej manualnie do falownika gdy awaria przeciążenie prądowe
   RUNG wire#powerrail
      Contact( "AlwaysTRUE" )
      Contact( "IsCurrentOverloadInverter" )
      Move(in := "dbtags_Sterowanie".SetupControlPompownia.CurrentMax_Manual_Hz, out1 => "dbdane".Manual_SV)
   END_RUNG
   // the same network as SCL:
   IF "AlwaysTRUE" AND "IsCurrentOverloadInverter" THEN
       "dbdane".Manual_SV := "dbtags_Sterowanie".SetupControlPompownia.CurrentMax_Manual_Hz;
   END_IF;
END_REGION

REGION Network 17: Ustawienie tymczasowych Hz
   // Ustawienie tymczasowej wartości Hz
   RUNG wire#powerrail
      Contact( "Tmp_Set_SV" )
      Move(in := "dbTable of value Hz".Static_1[15], out1 => "dbdane".Manual_SV)
   END_RUNG
   // the same network as SCL:
   IF "Tmp_Set_SV" THEN "dbdane".Manual_SV := "dbTable of value Hz".Static_1[15]; END_IF;
END_REGION

REGION Network 18: Ustawienie bitu sygnały tymczasowej wartości Hz
   // Gdy Hz zadawane z PID są mniejsze od 15.0 Hz a wartość bar mniejsza od zadanej i mniejsza od zera lub równa to ustaw wartość Hz tymczasową
   RUNG wire#powerrail
      I_Contact( "FirstScan" )
      I_Contact( "BarPress_Max" )
      I_Contact( "IsCurrentOverloadInverter" )
      Contact( "IEC_Timer_Reset_delay_DB".Q )
      { S7_Templates := "SrcType := Real" } LT_Contact(in1 := "dbdane".PV, in2 := "dbdane".Setpoint_SV)
      { S7_Templates := "SrcType := Real" } LE_Contact(in1 := "dbdane".OUT_PURE_Real, in2 := 15.0)
      S_Coil( "Tmp_Set_SV" )
   END_RUNG
   // the same network as SCL:
   IF NOT "FirstScan" AND NOT "BarPress_Max" AND NOT "IsCurrentOverloadInverter" AND "IEC_Timer_Reset_delay_DB".Q AND ("dbdane".PV < "dbdane".Setpoint_SV) AND ("dbdane".OUT_PURE_Real <= 15.0) THEN
       "Tmp_Set_SV" := TRUE;
   END_IF;
END_REGION

REGION Network 19: Reset znacznika ustawiania tymczasowej wartości Hz P1-P4
   RUNG wire#powerrail
      { S7_Templates := "SrcType := Real" } GE_Contact(in1 := "dbdane".OUT_PURE_Real, in2 := 16.0)
      wire#w1
      R_Coil( "Tmp_Set_SV" )
   END_RUNG
   RUNG wire#powerrail
      { S7_Templates := "SrcType := Real" } LE_Contact(in1 := "dbdane".PV, in2 := 0.0)
   END_RUNG wire#w1
   RUNG wire#powerrail
      Contact( "AlwaysTRUE" )
      { S7_Templates := "SrcType := Real" } GT_Contact(in1 := "dbdane".PV, in2 := "dbdane".Setpoint_SV)
   END_RUNG wire#w1
   // the same network as SCL:
   IF ("dbdane".OUT_PURE_Real >= 16.0) OR ("dbdane".PV <= 0.0) OR ("AlwaysTRUE" AND ("dbdane".PV > "dbdane".Setpoint_SV)) THEN
       "Tmp_Set_SV" := FALSE;
   END_IF;
END_REGION

REGION Network 20: Skalowanie wartości tymczasowych Hz to %QW P1-P4
   // "dane".Temp_SV - Tymczasowa wartość Hz  (30Hz)
   RUNG wire#powerrail
      Contact( "AlwaysTRUE" )
      Move(in := 8294, out1 => "dbdane".Temp_SV)
   END_RUNG
   // the same network as SCL:
   IF "AlwaysTRUE" THEN "dbdane".Temp_SV := 8294; END_IF;
END_REGION

REGION Network 21: Histerezas Reset Hz ustawionych manualnie
   RUNG wire#powerrail
      { S7_Templates := "SrcType := Real" } GE_Contact(in1 := "dbdane".OUT_PURE_Real, in2 := 10.0)
      { S7_Templates := "time_type := Time" } "IEC_Timer_Set_50Hz_DB".TON(pt := T#20S, et =>)
   END_RUNG
   // the same network as SCL:
   "IEC_Timer_Set_50Hz_DB".TON(IN := "dbdane".OUT_PURE_Real >= 10.0, PT := T#20S);
END_REGION

REGION Network 22: Reset znacznika płynnego przełaczenie Hz z tymczasowych na podawane z PID
   // Reset znacznika manualnego zadawania Hz
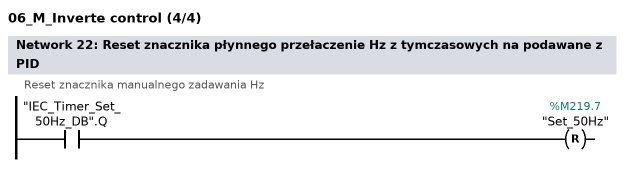
   RUNG wire#powerrail
      Contact( "IEC_Timer_Set_50Hz_DB".Q )
      R_Coil( "Set_50Hz" )
   END_RUNG
   // the same network as SCL:
   IF "IEC_Timer_Set_50Hz_DB".Q THEN "Set_50Hz" := FALSE; END_IF;
END_REGION
END_FUNCTION_BLOCK

FUNCTION_BLOCK "06_M_Network connection control"   // FB10, LAD
TITLE = Sterowanie stycznikiem sieć
{ S7_Optimized_Access := 'TRUE' }
AUTHOR : rtecmer
VERSION : 0.1
// Sterowanie stycznikiem sieć. Ustawianie znaczników setCMD_SM i setSUPV_SM które przekazywane są do funkcji FC3/FC1 DRV01 driver napędów. Następnie przekazywane jest do warstwy Hardware/ OUT gdzie ustawiane jest wyjście sterownika
// stored: AutoNumber true, IsIECCheckEnabled false, IsRetainMemResEnabled false, MemoryReserve 500, SetENOAutomatically false, UDAEnableTagReadback false
   VAR_INPUT
      IsReady_M : Bool;   // Gotowość napędu
      IsModeAut : Bool;   // Znacznik tryb pracy
      Time_Off_Inverter : Bool;   // Bit Q - timer blokowania stycznika falownika po wyłączeniu
      setMotor2 : Bool;   // Znacznik dodatkowa pompy nr1
      setMotor3 : Bool;   // Znacznik ustawienie dodatkowej 2
      setMotor4 : Bool;   // Znacznik ustawienie dodatkowej 3
      IsRunNetwork_M : Bool;   // Potwierdzenie pracy z sieci M
      CMD_A_NetworkM : Bool;   // Znacznik serowania awaryjnego napędem z sieci w wypadku awarii falownika
   END_VAR
   VAR_IN_OUT
      TimerStartNetworkContactor : TON_TIME;   // Opóżnienie załaczenia stycznika sieć
      setCMD_SM : Bool;   // Znacznik sterowania stycznikiem sieć
      Is_extras_K1_M_1 : Bool;   // Znacznik motor dodatkowy nr 1
      Is_extras_K2_M_1 : Bool;   // Znacznik motor dodatkowy nr 2
      Is_extras_K3_M_1 : Bool;   // Znacznik motor dodatkowy nr 3
      setSUPV_SM : Bool;   // Znacznik polecenia sterowania z sieci
      off_add_K1 : Bool;   // znacznik pomocniczy podczas selektrywnego wyłączeania dodatkowej pompy
      off_add_K2 : Bool := false;   // znacznik pomocniczy podczas selektrywnego wyłączeania dodatkowej pompy
      off_add_K3 : Bool := false;   // znacznik pomocniczy podczas selektrywnego wyłączeania dodatkowej pompy
   END_VAR
   VAR
      tmpOFFinverter { ExternalAccessible := 'False'; ExternalVisible := 'False'; ExternalWritable := 'False'} : Bool;   // wyłączenie od osiągnięcia 50Hz + czas zwłoki
      mem_activ_K1 { ExternalAccessible := 'False'; ExternalVisible := 'False'; ExternalWritable := 'False'} : Bool;   // pamięć załączennie jako dodatkowa
      mem_activ_K2 { ExternalAccessible := 'False'; ExternalVisible := 'False'; ExternalWritable := 'False'} : Bool;   // pamięć załączennie jako dodatkowa
      mem_activ_K3 { ExternalAccessible := 'False'; ExternalVisible := 'False'; ExternalWritable := 'False'} : Bool;   // pamięć załączennie jako dodatkowa
   END_VAR
   VAR_TEMP   // added for the SCL form of the ladder/FBD networks
      _w1 : Bool;
   END_VAR
BEGIN

REGION Network 1: Timer opóźnienie dołączenie stycznika sieci
   // Histereza na dołączenie stycznika sieć po pracy z falownika
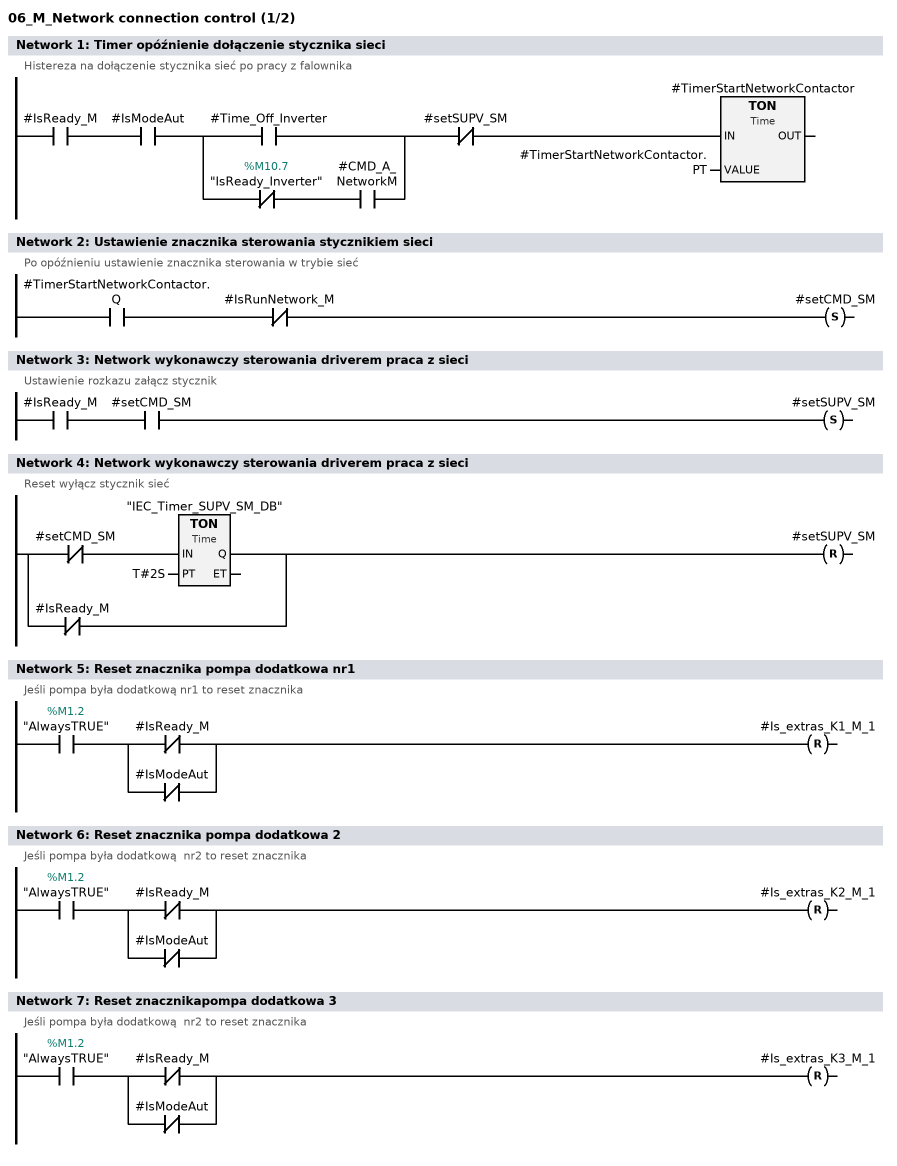
   #TimerStartNetworkContactor(IN := #IsReady_M AND #IsModeAut AND (#Time_Off_Inverter OR (NOT "IsReady_Inverter" AND #CMD_A_NetworkM)) AND NOT #setSUPV_SM, PT := #TimerStartNetworkContactor.PT);   // TON coil
END_REGION

REGION Network 2: Ustawienie znacznika sterowania stycznikiem sieci
   // Po opóźnieniu ustawienie znacznika sterowania w trybie sieć
   RUNG wire#powerrail
      Contact( #TimerStartNetworkContactor.Q )
      I_Contact( #IsRunNetwork_M )
      S_Coil( #setCMD_SM )
   END_RUNG
   // the same network as SCL:
   IF #TimerStartNetworkContactor.Q AND NOT #IsRunNetwork_M THEN #setCMD_SM := TRUE; END_IF;
END_REGION

REGION Network 3: Network wykonawczy sterowania driverem praca z sieci
   // Ustawienie rozkazu załącz stycznik
   RUNG wire#powerrail
      Contact( #IsReady_M )
      Contact( #setCMD_SM )
      S_Coil( #setSUPV_SM )
   END_RUNG
   // the same network as SCL:
   IF #IsReady_M AND #setCMD_SM THEN #setSUPV_SM := TRUE; END_IF;
END_REGION

REGION Network 4: Network wykonawczy sterowania driverem praca z sieci
   // Reset wyłącz stycznik sieć
   RUNG wire#powerrail
      I_Contact( #setCMD_SM )
      { S7_Templates := "time_type := Time" } "IEC_Timer_SUPV_SM_DB".TON(pt := T#2S, et =>)
      wire#w1
      R_Coil( #setSUPV_SM )
   END_RUNG
   RUNG wire#powerrail
      I_Contact( #IsReady_M )
   END_RUNG wire#w1
   // the same network as SCL:
   "IEC_Timer_SUPV_SM_DB".TON(IN := NOT #setCMD_SM, PT := T#2S);
   IF "IEC_Timer_SUPV_SM_DB".Q OR NOT #IsReady_M THEN #setSUPV_SM := FALSE; END_IF;
END_REGION

REGION Network 5: Reset znacznika pompa dodatkowa nr1
   // Jeśli pompa była dodatkową nr1 to reset znacznika
   RUNG wire#powerrail
      Contact( "AlwaysTRUE" )
      wire#w1
      I_Contact( #IsReady_M )
      wire#w2
      R_Coil( #Is_extras_K1_M_1 )
   END_RUNG
   RUNG wire#w1
      I_Contact( #IsModeAut )
   END_RUNG wire#w2
   // the same network as SCL:
   IF "AlwaysTRUE" AND (NOT #IsReady_M OR NOT #IsModeAut) THEN #Is_extras_K1_M_1 := FALSE; END_IF;
END_REGION

REGION Network 6: Reset znacznika pompa dodatkowa 2
   // Jeśli pompa była dodatkową  nr2 to reset znacznika
   RUNG wire#powerrail
      Contact( "AlwaysTRUE" )
      wire#w1
      I_Contact( #IsReady_M )
      wire#w2
      R_Coil( #Is_extras_K2_M_1 )
   END_RUNG
   RUNG wire#w1
      I_Contact( #IsModeAut )
   END_RUNG wire#w2
   // the same network as SCL:
   IF "AlwaysTRUE" AND (NOT #IsReady_M OR NOT #IsModeAut) THEN #Is_extras_K2_M_1 := FALSE; END_IF;
END_REGION

REGION Network 7: Reset znacznikapompa dodatkowa 3
   // Jeśli pompa była dodatkową  nr2 to reset znacznika
   RUNG wire#powerrail
      Contact( "AlwaysTRUE" )
      wire#w1
      I_Contact( #IsReady_M )
      wire#w2
      R_Coil( #Is_extras_K3_M_1 )
   END_RUNG
   RUNG wire#w1
      I_Contact( #IsModeAut )
   END_RUNG wire#w2
   // the same network as SCL:
   IF "AlwaysTRUE" AND (NOT #IsReady_M OR NOT #IsModeAut) THEN #Is_extras_K3_M_1 := FALSE; END_IF;
END_REGION

REGION Network 8: Reset Znacznika sterowania w trybie sieć
   // Gdy regulator PID ustawi szybkie wyłaczenie pompy dodatkowej nr 1, nr 2, nr 3 to następuje resetowania znacznika pracy pompy dodatkowej
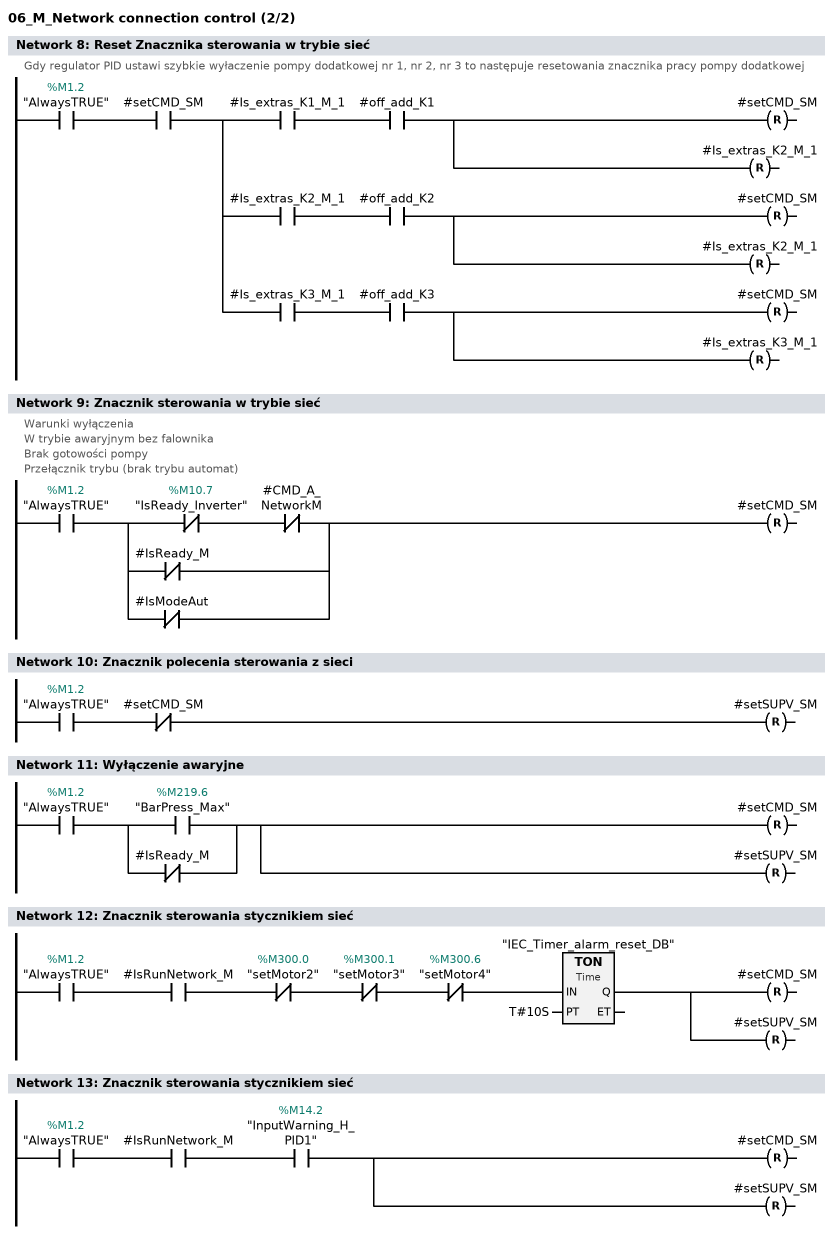
   RUNG wire#powerrail
      Contact( "AlwaysTRUE" )
      Contact( #setCMD_SM )
      wire#w1
      Contact( #Is_extras_K1_M_1 )
      Contact( #off_add_K1 )
      wire#w2
      R_Coil( #setCMD_SM )
   END_RUNG
   RUNG wire#w2
      R_Coil( #Is_extras_K2_M_1 )
   END_RUNG
   RUNG wire#w1
      Contact( #Is_extras_K2_M_1 )
      Contact( #off_add_K2 )
      wire#w3
      R_Coil( #setCMD_SM )
   END_RUNG
   RUNG wire#w3
      R_Coil( #Is_extras_K2_M_1 )
   END_RUNG
   RUNG wire#w1
      Contact( #Is_extras_K3_M_1 )
      Contact( #off_add_K3 )
      wire#w4
      R_Coil( #setCMD_SM )
   END_RUNG
   RUNG wire#w4
      R_Coil( #Is_extras_K3_M_1 )
   END_RUNG
   // the same network as SCL:
   #_w1 := "AlwaysTRUE" AND #setCMD_SM;
   IF #_w1 AND #Is_extras_K1_M_1 AND #off_add_K1 THEN
       #setCMD_SM := FALSE;
       #Is_extras_K2_M_1 := FALSE;
   END_IF;
   IF #_w1 AND #Is_extras_K2_M_1 AND #off_add_K2 THEN
       #setCMD_SM := FALSE;
       #Is_extras_K2_M_1 := FALSE;
   END_IF;
   IF #_w1 AND #Is_extras_K3_M_1 AND #off_add_K3 THEN
       #setCMD_SM := FALSE;
       #Is_extras_K3_M_1 := FALSE;
   END_IF;
END_REGION

REGION Network 9: Znacznik sterowania w trybie sieć
   // Warunki wyłączenia 
   // W trybie awaryjnym bez falownika
   // Brak gotowości pompy
   // Przełącznik trybu (brak trybu automat)
   RUNG wire#powerrail
      Contact( "AlwaysTRUE" )
      wire#w1
      I_Contact( "IsReady_Inverter" )
      I_Contact( #CMD_A_NetworkM )
      wire#w2
      R_Coil( #setCMD_SM )
   END_RUNG
   RUNG wire#w1
      I_Contact( #IsReady_M )
   END_RUNG wire#w2
   RUNG wire#w1
      I_Contact( #IsModeAut )
   END_RUNG wire#w2
   // the same network as SCL:
   IF "AlwaysTRUE" AND ((NOT "IsReady_Inverter" AND NOT #CMD_A_NetworkM) OR NOT #IsReady_M OR NOT #IsModeAut) THEN
       #setCMD_SM := FALSE;
   END_IF;
END_REGION

REGION Network 10: Znacznik polecenia sterowania z sieci
   RUNG wire#powerrail
      Contact( "AlwaysTRUE" )
      I_Contact( #setCMD_SM )
      R_Coil( #setSUPV_SM )
   END_RUNG
   // the same network as SCL:
   IF "AlwaysTRUE" AND NOT #setCMD_SM THEN #setSUPV_SM := FALSE; END_IF;
END_REGION

REGION Network 11: Wyłączenie awaryjne
   RUNG wire#powerrail
      Contact( "AlwaysTRUE" )
      wire#w1
      Contact( "BarPress_Max" )
      wire#w2
      R_Coil( #setCMD_SM )
   END_RUNG
   RUNG wire#w1
      I_Contact( #IsReady_M )
   END_RUNG wire#w2
   RUNG wire#w2
      R_Coil( #setSUPV_SM )
   END_RUNG
   // the same network as SCL:
   IF "AlwaysTRUE" AND ("BarPress_Max" OR NOT #IsReady_M) THEN
       #setCMD_SM := FALSE;
       #setSUPV_SM := FALSE;
   END_IF;
END_REGION

REGION Network 12: Znacznik sterowania stycznikiem sieć
   RUNG wire#powerrail
      Contact( "AlwaysTRUE" )
      Contact( #IsRunNetwork_M )
      I_Contact( "setMotor2" )
      I_Contact( "setMotor3" )
      I_Contact( "setMotor4" )
      { S7_Templates := "time_type := Time" } "IEC_Timer_alarm_reset_DB".TON(pt := T#10S, et =>)
      wire#w1
      R_Coil( #setCMD_SM )
   END_RUNG
   RUNG wire#w1
      R_Coil( #setSUPV_SM )
   END_RUNG
   // the same network as SCL:
   "IEC_Timer_alarm_reset_DB".TON(IN := "AlwaysTRUE" AND #IsRunNetwork_M AND NOT "setMotor2" AND NOT "setMotor3" AND NOT "setMotor4",
                           PT := T#10S);
   IF "IEC_Timer_alarm_reset_DB".Q THEN
       #setCMD_SM := FALSE;
       #setSUPV_SM := FALSE;
   END_IF;
END_REGION

REGION Network 13: Znacznik sterowania stycznikiem sieć
   RUNG wire#powerrail
      Contact( "AlwaysTRUE" )
      Contact( #IsRunNetwork_M )
      Contact( "InputWarning_H_PID1" )
      wire#w1
      R_Coil( #setCMD_SM )
   END_RUNG
   RUNG wire#w1
      R_Coil( #setSUPV_SM )
   END_RUNG
   // the same network as SCL:
   IF "AlwaysTRUE" AND #IsRunNetwork_M AND "InputWarning_H_PID1" THEN
       #setCMD_SM := FALSE;
       #setSUPV_SM := FALSE;
   END_IF;
END_REGION
END_FUNCTION_BLOCK

FUNCTION "04_A_OUT" : Void
TITLE = OUT 
{ S7_Optimized_Access := 'TRUE' }
AUTHOR : rtecmer
VERSION : 0.1
//Mapowamie i wyzwalanie wyjść 

BEGIN
	(*
	//=============================================================================
	//(JZWiK S.A Radosław Tecmer)
	//(c)Copyright (2021) All Rights Reserved
	//-----------------------------------------------------------------------------
	//Testowane z:   (system docelowy z  FW 4.4)
	//Pakiet inżynierski:   TIA Portal (V14 Sp1 Update 9)
	//Ograniczenia:  ( - )
	//Wymagania:  (minimalne S7-1200 CPU 1215C FW 4.2 .)
	//Funkcjonalnośc: (Sterowania napędami poprzez przekazanie wartości na 
	//                  wyjście sterownika )
	//-----------------------------------------------------------------------------
	//Zmainy wprowadzone:
	//Wersja  Data       Osoba wprowadzająca zmiany - ekspert
	//01.00.00 19.01.2022 (Tecmer Radosław - twórca) Pieresza wersja 01.00.00
	//=============================================================================
	*)
	
	
	
	REGION Sygnalizacja Awarii
	  
	  // Wyjścia przekaźnikowe sygnalizacja awarii
	  //Pomp Zasuw Falownika Soft-start
	  "Q0.7" := "CMD_faultInverter";
	  "Q0.4" := "CMD_faultP1";
	  "Q0.5" := "CMD_faultP2";
	  "Q2.6" := "CMD_faultP3";
	  "Q2.7" := "CMD_faultP4";
	  
	END_REGION
	
	REGION "inverter"
	  // Start stop inverter
	  IF "CMD_start_stop_inverter" THEN
	    //Jeśli tylko jeden stycznik dla folowika dołączony
	    IF ("IsRunInverter_P1" XOR "IsRunInverter_P2" XOR "IsRunInverter_P3" XOR "IsRunInverter_P4") AND
	      NOT ("IsRunInverter_P1" AND "IsRunInverter_P2") AND
	      NOT ("IsRunInverter_P1" AND "IsRunInverter_P3") AND
	      NOT ("IsRunInverter_P1" AND "IsRunInverter_P4") AND
	      NOT ("IsRunInverter_P2" AND "IsRunInverter_P3") AND
	      NOT ("IsRunInverter_P2" AND "IsRunInverter_P4") AND
	      NOT ("IsRunInverter_P3" AND "IsRunInverter_P4") AND
	      NOT "IsCurrentOverloadInverter"
	      
	    THEN
	      // 
	      "Q0.6" := TRUE;
	    ELSE
	      "Q0.6" := FALSE;
	      ;
	    END_IF;
	  ELSE
	    "Q0.6" := FALSE;
	    ;
	  END_IF;
	  
	  // resset alarmu falownika
	  "Q1.1" := "resetAlarm_Inverter";
	  
	END_REGION
	
	
	REGION Styczniki P1
	  // Uruchamianie wyjść sterujących stycznik pompoy falownik, sieć
	  IF "CMD_inverter_P1" THEN
	    // 
	    IF NOT ("IsRunInverter_P2") AND NOT ("IsRunInverter_P3") AND NOT ("IsRunInverter_P4")AND NOT "IsCurrentOverloadInverter" THEN
	      // 
	      "Q0.0" := True;
	    ELSE
	      "Q0.0" := FALSE;
	      ;
	    END_IF;
	  ELSE
	    "Q0.0" := FALSE;
	    ;
	  END_IF;
	  
	  
	  "Q0.1" := "CMD_network_P1";
	  
	  
	 
	END_REGION
	
	REGION Styczniki P2
	  // Uruchamianie wyjść sterujących stycznik pompoy falownik, sieć
	  IF "CMD_inverter_P2" THEN
	    // 
	    IF NOT ("IsRunInverter_P1") AND NOT ("IsRunInverter_P3") AND NOT ("IsRunInverter_P4")AND NOT "IsCurrentOverloadInverter" THEN
	      // 
	      "Q0.2" := True;
	    ELSE
	      "Q0.2" := FALSE;
	      ;
	    END_IF;
	  ELSE
	    "Q0.2" := FALSE;
	    ;
	  END_IF;
	
	  
	  "Q0.3" := "CMD_network_P2";
	  
	  
	  
	END_REGION
	
	REGION Styczniki P3
	  // Uruchamianie wyjść sterujących stycznik pompoy falownik, sieć
	  IF "CMD_inverter_P3" THEN
	    // 
	    IF NOT ("IsRunInverter_P1") AND NOT ("IsRunInverter_P2") AND NOT ("IsRunInverter_P4") AND NOT "IsCurrentOverloadInverter" THEN
	      // 
	      "Q0.4" := True;
	    ELSE
	      "Q0.4" := FALSE;
	      ;
	    END_IF;
	  ELSE
	    "Q0.4" := FALSE;
	    ;
	  END_IF;
	  
	  
	  "Q0.5" := "CMD_network_P3";
	  
	  
	  
	END_REGION
	
	
	
	REGION Zasuwa Z11
	  // Przekazanie wartości
	  //Otwieranie
	  "Q2.0" := "CMD_Open_Z11";
	  //Zamykanie
	  "Q2.1" := "CMD_Close_Z11";
	
	  
	END_REGION
	
	
	  
	
	
	
	
	
	
	
	
	
	
	 
	
	
	
	
	 
	 
	
	 
	 
	 
END_FUNCTION

FUNCTION "08_M_Conroll_from_ModbusRTU" : Void
{ S7_Optimized_Access := 'TRUE' }
AUTHOR : rtecmer
VERSION : 0.1

BEGIN
	(*
	//=============================================================================
	//(JZWiK S.A Radosław Tecmer)
	//(c)Copyright (2021) All Rights Reserved
	//-----------------------------------------------------------------------------
	//Testowane z:   (system docelowy z  FW 4.2)
	//Pakiet inżynierski:   TIA Portal (V14 Sp1 Update 9)
	//Ograniczenia:  ( - )
	//Wymagania:  (minimalne S7-1200 CPU 1214 FW 3.2 .)
	//Funkcjonalnośc: (Przesuniecie bajtów (podobnie do funkcji SWAP) 
	//                  i przekazanie do bloku danych pomiary z przepływomierza )
	//-----------------------------------------------------------------------------
	//Zmainy wprowadzone:
	//Wersja  Data       Osoba wprowadzająca zmiany - ekspert
	//01.00.00 17.11.2021 (Tecmer Radosław - twórca) Pieresza wersja 01.00.00
	//=============================================================================
	*)
	
	
	
	REGION Q1 przepływomierz
	  // Adres 0 - bierzący przepływ
	 
	 
	  "dbdane".Wielkość_przeływu_Q1 := "dbModbusRTU_Reg"."Przepływomierz nr1 pompownia".ID6_przeływu_VF_Adres_0;
	  
	  // Adres 2 - Licznik_objętość_VF
	 
	  
	  "dbdane".Licznik_objętość_VF_Q1 := "dbModbusRTU_Reg"."Przepływomierz nr1 pompownia".ID6_objętość_VF_Adres_2;
	  
	  // Adres 4- stan bierzący licznika objetości w stecz VR
	  
	  
	  "dbdane".Licznik_objętość_VR_Q1 := "dbModbusRTU_Reg"."Przepływomierz nr1 pompownia"."ID6_objętośc RF_Adres_4";
	  
	 
	END_REGION
	
	
	
	  
	  
	  
	  
	  
	  
	
	
END_FUNCTION

FUNCTION_BLOCK "01_E_Alarm_min_bar_empty_tanks"
TITLE = Start procedury awarujnego pompowania
{ S7_Optimized_Access := 'TRUE' }
AUTHOR : rt69
VERSION : 0.1
//Funkcja rozpoczyna procedurę awaryjnego sterowaia zasilaniem na magistralę 
   VAR_OUTPUT 
      bit_alarm_magistrala_min { ExternalAccessible := 'False'; ExternalVisible := 'False'; ExternalWritable := 'False'} : Bool := false;   // bit alarmmagistrala awaria niskie ciśnienie
   END_VAR

   VAR_IN_OUT 
      bit_off_alarm_niskie_magistrala { ExternalAccessible := 'False'; ExternalVisible := 'False'; ExternalWritable := 'False'} : Bool;   // bit koniec alarmu niskie bar magistrala
      "tempStrategia Pompownia" : Int := 16#0;   // przechwycone słowo strategii pompownia
      "actStrategia Pompownia" : Int;   // Słowo reprezentujące strategie sterowania pompownią (wyłączona , przetłaczanie , dosilanie,automat)
   END_VAR

   VAR 
      memTriger_Strategia { ExternalAccessible := 'False'; ExternalVisible := 'False'; ExternalWritable := 'False'} : Bool;   // pamięć zbocza
      bit_normalne_magistrala { ExternalAccessible := 'False'; ExternalVisible := 'False'; ExternalWritable := 'False'} : Bool;   // bit detekcjinormalnego cisnienia magistrala
      bit_niskie_magistrala { ExternalAccessible := 'False'; ExternalVisible := 'False'; ExternalWritable := 'False'} : Bool;   // bit detekcji niskiego cisnienia magistrala
      memFalling_allarm : Bool;
   END_VAR


BEGIN
	(*
	//=============================================================================
	//(JZWiK S.A Radosław Tecmer)
	//(c)Copyright (2021) All Rights Reserved
	//-----------------------------------------------------------------------------
	//Testowane z:   (system docelowy z  FW 4.4)
	//Pakiet inżynierski:   TIA Portal (V14 Sp1 Update 9)
	//Ograniczenia:  ( - )
	//Wymagania:  (minimalne S7-1200 CPU 1215C FW 4.2 .)
	//Funkcjonalnośc: (Funkcja ustawia lub kasuje bit alarmu od niskiego
	                   ciśnieia na magistrali - od czujnika B5)
	//-----------------------------------------------------------------------------
	//Zmainy wprowadzone:
	//Wersja  Data       Osoba wprowadzająca zmiany - ekspert
	//01.00.00 17.11.2021 (Tecmer Radosław - twórca) Pieresza wersja 01.00.00
	//=============================================================================
	*)
	
	
	
	
	IF "dbHoldRegSlave_to_MT101".instB5bar_act < "dbHoldRegSlave_to_MT101".instSetBarMinB9
	  AND "dbHoldRegSlave_to_MT101".instSygSter_2 <> 0 AND
	  ("dbHoldRegSlave_to_MT101".instLevelTank1 <= 50 AND "dbHoldRegSlave_to_MT101".instLevelTank2 <= 50 AND "dbHoldRegSlave_to_MT101".instLevelTank3 <= 50) THEN
	  // Statement section IF
	  // Ustaw bit za niskie ciśnienie
	  #bit_niskie_magistrala := TRUE;
	ELSE
	  ;
	END_IF;
	
	IF "dbHoldRegSlave_to_MT101".instB5bar_act < "dbHoldRegSlave_to_MT101".instSetBarMinB9
	  AND "dbHoldRegSlave_to_MT101".instSygSter_2 = 0
	  
	THEN
	  // Statement section IF
	  // Ustaw bit za niskie ciśnienie
	  #bit_niskie_magistrala := TRUE;
	ELSE
	   ;
	END_IF;
	
	
	
	"R_TRIG_DB_przechwycenie_strategii"(CLK := #bit_niskie_magistrala,
	                                    Q => #memTriger_Strategia);
	IF #memTriger_Strategia THEN
	  // zatrzaśniecie przechwyconą strategię 
	  #"tempStrategia Pompownia" := #"actStrategia Pompownia";
	  IF #"tempStrategia Pompownia" = 0 THEN
	    // to wpisz domyślną 2
	    #"tempStrategia Pompownia" := 3
	    ;
	  END_IF;
	END_IF;
	  
	
	
	
	"F_TRIG_DB_przechwycenie_powrotu_bar_valueTanks"(CLK := #bit_niskie_magistrala,
	                                                 Q => #memFalling_allarm);
	IF #memFalling_allarm THEN
	  // przekazanie zatrzaśniętej wartości po powrocie poprawnych warunków w sieci zasilającej/ zbiornikach 
	  #"tempStrategia Pompownia" := #"actStrategia Pompownia";
	  IF #"tempStrategia Pompownia" = 0 THEN
	    // to wpisz domyślną 2
	    #"tempStrategia Pompownia" := 3
	    ;
	  END_IF;
	  
	  ;
	END_IF;
	
	
	// Histereza na ustawienie alarmu "niskie ćiśnienie na magistrali"
	"IEC_Timer_AlarmMagistrala_Niskie_DB".TON(IN := #bit_niskie_magistrala,
	                                          PT := T#30S,
	                                          Q => #bit_alarm_magistrala_min);
	
	
	
	
	// Sprawdzanie powrotu zasilania z magistrali czujnik B5 i (zbiorniki)
	IF "dbHoldRegSlave_to_MT101".instB5bar_act > 1.0 OR
	  "dbHoldRegSlave_to_MT101".instLevelTank1 >= 250 OR
	  "dbHoldRegSlave_to_MT101".instLevelTank2 >= 250
	THEN
	  // Ustaw bit  normalne ciśnienie
	  #bit_normalne_magistrala := TRUE;
	  
	ELSE
	  #bit_normalne_magistrala := FALSE;
	  ;
	END_IF;
	
	
	//Histerez na powrót normalnego zasilania z magistrali
	"IEC_Timer_resetAlarmMagistrala_Niskie_DB".TON(IN := #bit_normalne_magistrala,
	                                               Q => #bit_off_alarm_niskie_magistrala,
	                                               PT := T#1M);
	
	
	IF #bit_off_alarm_niskie_magistrala THEN
	  // kasuj alarm niskie magistrala
	  #bit_niskie_magistrala := FALSE;
	END_IF;
	
	
END_FUNCTION_BLOCK

FUNCTION_BLOCK "06_M_Initialization of start values"
TITLE = Setup Write Parameters_KDN
{ S7_Optimized_Access := 'TRUE' }
AUTHOR : rtecmer
VERSION : 0.1
//Pobranie parametrów technologicznych i przekazanie ich do instancji "tags" w celu zachowania i wprowadzeni po resecie PLC
   VAR 
      TimeHz_DInt { ExternalAccessible := 'False'; ExternalVisible := 'False'; ExternalWritable := 'False'} : DInt;
   END_VAR


BEGIN
	(*
	//=============================================================================
	//(JZWiK S.A Radosław Tecmer)
	//(c)Copyright (2021) All Rights Reserved
	//-----------------------------------------------------------------------------
	//Testowane z:   (system docelowy z  FW 4.2)
	//Pakiet inżynierski:   TIA Portal (V14 Sp1 Update 9)
	//Ograniczenia:  ( - )
	//Wymagania:  (minimalne S7-1200 CPU 1214 FW 3.2 .)
	//Funkcjonalnośc: (Przekazanie warotości ostatnio wpisanych do instancji "tags 
	                   w celu przechowania danych. W czasie restartu CPU będą wczytywane
	                   do parametrów sterowania  )
	//-----------------------------------------------------------------------------
	//Zmainy wprowadzone:
	//Wersja  Data       Osoba wprowadzająca zmiany - ekspert
	//01.00.00 17.11.2021 (Tecmer Radosław - twórca) Pieresza wersja 01.00.00
	//=============================================================================
	*)
	
	
	REGION Sterowanie 
	  
	  //Czas oczekiwania na 50Hz 
	  "dbdane".TMR_Hz := DINT_TO_TIME(#TimeHz_DInt * "MS_TO_S");
	  
	  //Tryb pracy pompowni 
	  "dbtags_Sterowanie".SetupControlPompownia.Switch_Aut_Rem_Pompy := "dbmanagement".sterowanie_1.tryb_automat;
	  
	  //strategi pracy pompowni
	  "dbdane".Switch_model_control_P1P4 := "dbHoldRegSlave_to_MT101".instSygSter_1;
	  //strategia sterowaia zbiornikami
	  "dbdane".Switch_model_control_Tanks := "dbHoldRegSlave_to_MT101".instSygSter_2;
	  
	  //kasowanie alarmów napędów
	  "dbtags_Sterowanie"."Paramaetry _Zbiorniki".rez_alarm_napędów := "dbHoldRegSlave_to_MT101".instClearFault1;
	  
	  // zadane ciśnieniea
	 
	  "dbtags_Sterowanie".SetupControlPompownia.set_barDN225_B6 := "dbHoldRegSlave_to_MT101".instSetbarDN225_B6;
	  
	  // zadane min ciśnienie magistrala
	  "dbtags_Sterowanie".SetupControlPompownia.setBarMinMainLine := "dbHoldRegSlave_to_MT101".instSetBarMinB9;
	  
	  // maksymalny dopuszczalny prąd falownika
	  
	  
	END_REGION
	
	REGION Z11 Z12 Status
	  // Przekazanie do instancji pamięci parametrów
	  IF %DB10.DBX118.7 = 1 THEN
	    // Gdy praca Auto ustaw
	    "dbtags_Sterowanie".SetupControlPompownia.Z11_Status := 33924;
	  ELSE
	    "dbtags_Sterowanie".SetupControlPompownia.Z11_Status := 0;
	  END_IF;
	  
	  IF %DB10.DBX120.7 = 1  THEN
	    // gdy praca Auto ustaw
	    "dbtags_Sterowanie".SetupControlPompownia.Z12_Status := 33924;
	  ELSE
	    "dbtags_Sterowanie".SetupControlPompownia.Z12_Status := 0;
	  END_IF;
	  
	 
	  
	  
	END_REGION
	
	REGION Parametry nastaw zbiorników 
	  // 
	  "dbtags_Sterowanie"."Paramaetry _Zbiorniki".set_poziom_napełniania:= "dbHoldRegSlave_to_MT101".instLevelSetFilling ;
	  "dbtags_Sterowanie"."Paramaetry _Zbiorniki".set_poziom_opróżniania:= "dbHoldRegSlave_to_MT101".instLevelSetEmptying ;
	  "dbtags_Sterowanie"."Paramaetry _Zbiorniki".set_strategia_sterowania := "dbHoldRegSlave_to_MT101".instSygSter_1;
	  "dbtags_Sterowanie"."Paramaetry _Zbiorniki".set_sterowanie_cyklem:= "dbHoldRegSlave_to_MT101".instSygSter_2 ;
	 
	  "dbtags_Sterowanie"."Paramaetry _Zbiorniki".set_bity_sterowania_napęami_1 := "dbHoldRegSlave_to_MT101".instControllDrivers_1;
	  "dbtags_Sterowanie"."Paramaetry _Zbiorniki".set_bity_sterowania_napęami_2 := "dbHoldRegSlave_to_MT101".instControllDrivers_2;
	  "dbtags_Sterowanie"."Paramaetry _Zbiorniki".set_bity_tryb_napędów_1 := "dbHoldRegSlave_to_MT101".instConrol_ManAut_1;
	  "dbtags_Sterowanie"."Paramaetry _Zbiorniki".set_bity_tryb_napędów_2 := "dbHoldRegSlave_to_MT101".instConrol_ManAut_2;
	  //Czasy
	  "dbtags_Sterowanie".Zbiorniki_Godziny.start_napełnianie.HOUR := "dbHoldRegSlave_to_MT101".instHourStart_Filling;
	  "dbtags_Sterowanie".Zbiorniki_Godziny.start_napełnianie.MINUTE := "dbHoldRegSlave_to_MT101".instMinutStart_Filling;
	  "dbtags_Sterowanie".Zbiorniki_Godziny.start_napełnianie.SECOND := 0;
	  
	  "dbtags_Sterowanie".Zbiorniki_Godziny.Stop_napełnianie.HOUR := "dbHoldRegSlave_to_MT101".instHourStop_Filling;
	  "dbtags_Sterowanie".Zbiorniki_Godziny.Stop_napełnianie.MINUTE := "dbHoldRegSlave_to_MT101".instMinutStopt_Filling;
	  "dbtags_Sterowanie".Zbiorniki_Godziny.Stop_napełnianie.SECOND := 0;
	  
	
	  
	  
	  
	  
	END_REGION
	
	
	
END_FUNCTION_BLOCK

ORGANIZATION_BLOCK "Cyclic interrupt"   // OB30, LAD, CyclicInterrupt
{ S7_Optimized_Access := 'TRUE' }
AUTHOR : RTecmer
VERSION : 0.1
// stored: AutoNumber true, IsIECCheckEnabled false, SetENOAutomatically false
   VAR_TEMP
      Temp_SV_Int : Int;
      PV_Temp : Real;
      Temp_1 : Real;
   END_VAR
   VAR_TEMP   // added for the SCL form of the ladder/FBD networks
      _w1 : Bool;
      _w2 : Bool;
   END_VAR
BEGIN

REGION Network 1: Wyłączenie wejścia pradowego w regulatorze PID
   // Przełączenie na Input PID  (wejście wartościci zadanej) wyłaczenie wejścia prądowego input_PER
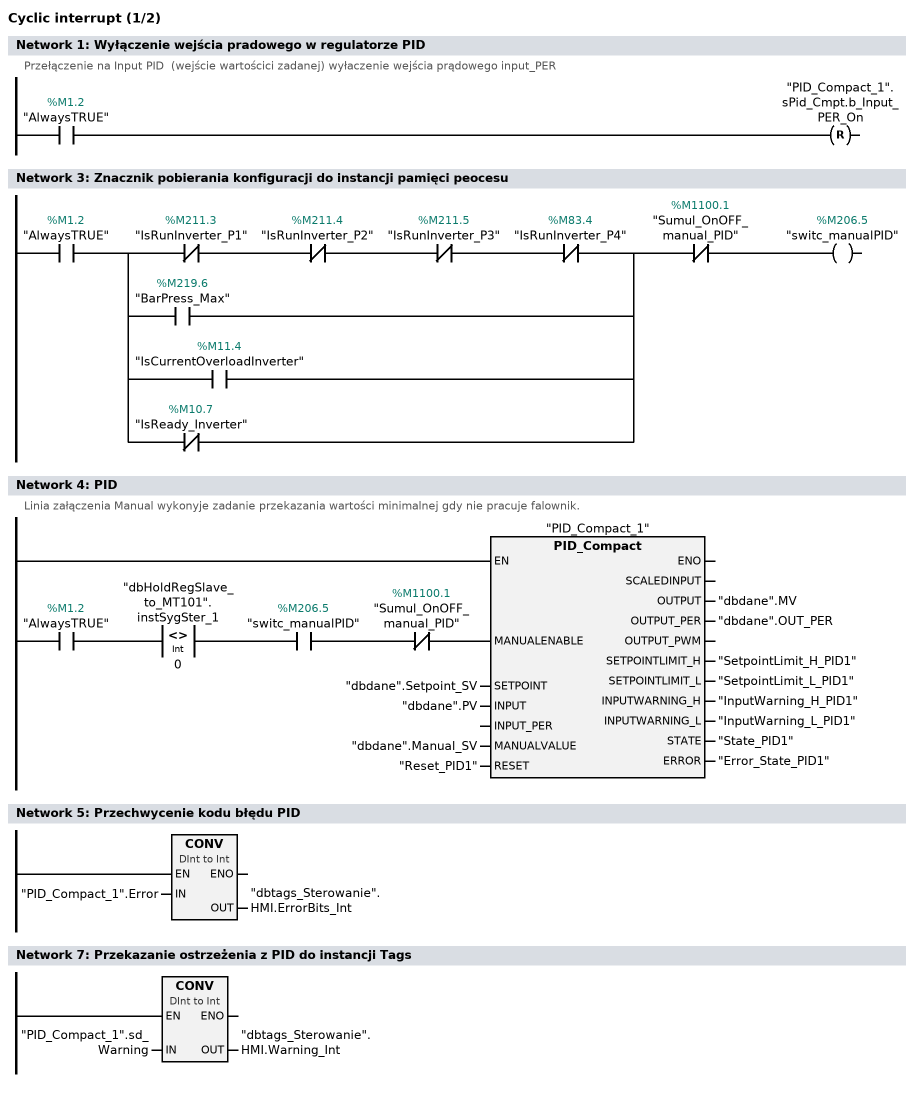
   RUNG wire#powerrail
      Contact( "AlwaysTRUE" )
      R_Coil( "PID_Compact_1".sPid_Cmpt.b_Input_PER_On )
   END_RUNG
   // the same network as SCL:
   IF "AlwaysTRUE" THEN "PID_Compact_1".sPid_Cmpt.b_Input_PER_On := FALSE; END_IF;
END_REGION

REGION Network 2: Skalowanie wartośc pressure oxygen
   // Przetwornik ciśnienia (0-1bar) 
   // !!!!!! Znienić po zamontowaniu właściwego !!!!!!! 
   // obecnie czujnik 10 bar
END_REGION

REGION Network 3: Znacznik pobierania konfiguracji do instancji pamięci peocesu
   RUNG wire#powerrail
      Contact( "AlwaysTRUE" )
      wire#w1
      I_Contact( "IsRunInverter_P1" )
      I_Contact( "IsRunInverter_P2" )
      I_Contact( "IsRunInverter_P3" )
      I_Contact( "IsRunInverter_P4" )
      wire#w2
      I_Contact( "Sumul_OnOFF_manual_PID" )
      Coil( "switc_manualPID" )
   END_RUNG
   RUNG wire#w1
      Contact( "BarPress_Max" )
   END_RUNG wire#w2
   RUNG wire#w1
      Contact( "IsCurrentOverloadInverter" )
   END_RUNG wire#w2
   RUNG wire#w1
      I_Contact( "IsReady_Inverter" )
   END_RUNG wire#w2
   // the same network as SCL:
   "switc_manualPID" := "AlwaysTRUE" AND ((NOT "IsRunInverter_P1" AND NOT "IsRunInverter_P2" AND NOT "IsRunInverter_P3" AND NOT "IsRunInverter_P4") OR "BarPress_Max" OR "IsCurrentOverloadInverter" OR NOT "IsReady_Inverter") AND NOT "Sumul_OnOFF_manual_PID";
END_REGION

REGION Network 4: PID
   // Linia załączenia Manual wykonyje zadanie przekazania wartości minimalnej gdy nie pracuje falownik.
   RUNG wire#powerrail
      "PID_Compact_1".PID_Compact(ManualEnable := wire#w1, Setpoint := "dbdane".Setpoint_SV, Input := "dbdane".PV, Input_PER :=, ManualValue := "dbdane".Manual_SV, Reset := "Reset_PID1", ScaledInput =>, Output => "dbdane".MV, Output_PER => "dbdane".OUT_PER, Output_PWM =>, SetpointLimit_H => "SetpointLimit_H_PID1", SetpointLimit_L => "SetpointLimit_L_PID1", InputWarning_H => "InputWarning_H_PID1", InputWarning_L => "InputWarning_L_PID1", State => "State_PID1", Error => "Error_State_PID1")
   END_RUNG
   RUNG wire#powerrail
      Contact( "AlwaysTRUE" )
      { S7_Templates := "SrcType := Int" } NE_Contact(in1 := "dbHoldRegSlave_to_MT101".instSygSter_1, in2 := 0)
      Contact( "switc_manualPID" )
      I_Contact( "Sumul_OnOFF_manual_PID" )
   END_RUNG wire#w1
   // the same network as SCL:
   "PID_Compact_1"(ManualEnable := "AlwaysTRUE" AND ("dbHoldRegSlave_to_MT101".instSygSter_1 <> 0) AND "switc_manualPID" AND NOT "Sumul_OnOFF_manual_PID",   // PID_Compact
                   Setpoint := "dbdane".Setpoint_SV,
                   Input := "dbdane".PV,
                   ManualValue := "dbdane".Manual_SV,
                   Reset := "Reset_PID1",
                   Output => "dbdane".MV,
                   Output_PER => "dbdane".OUT_PER,
                   SetpointLimit_H => "SetpointLimit_H_PID1",
                   SetpointLimit_L => "SetpointLimit_L_PID1",
                   InputWarning_H => "InputWarning_H_PID1",
                   InputWarning_L => "InputWarning_L_PID1",
                   State => "State_PID1",
                   Error => "Error_State_PID1");
END_REGION

REGION Network 5: Przechwycenie kodu błędu PID
   RUNG wire#powerrail
      { S7_Templates := "[SrcType := DInt, DestType := Int]"; S7_GenerateENO := "TRUE" } Convert(in := "PID_Compact_1".Error, out => "dbtags_Sterowanie".HMI.ErrorBits_Int)
   END_RUNG
   // the same network as SCL:
   "dbtags_Sterowanie".HMI.ErrorBits_Int := DINT_TO_INT("PID_Compact_1".Error);
END_REGION

REGION Network 7: Przekazanie ostrzeżenia z PID do instancji Tags
   RUNG wire#powerrail
      { S7_Templates := "[SrcType := DInt, DestType := Int]"; S7_GenerateENO := "TRUE" } Convert(in := "PID_Compact_1".sd_Warning, out => "dbtags_Sterowanie".HMI.Warning_Int)
   END_RUNG
   // the same network as SCL:
   "dbtags_Sterowanie".HMI.Warning_Int := DINT_TO_INT("PID_Compact_1".sd_Warning);
END_REGION

REGION Network 8: PID error reset
   // Reset PID od błędu
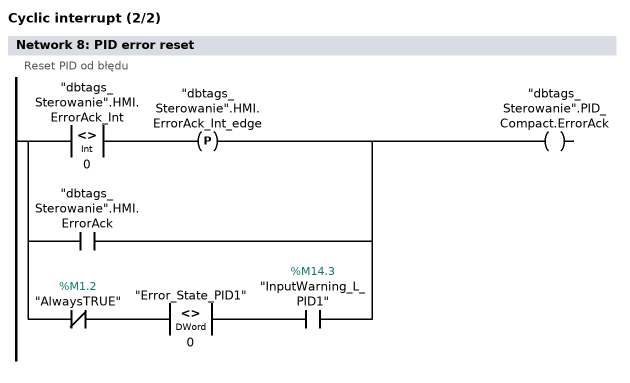
   RUNG wire#powerrail
      { S7_Templates := "SrcType := Int" } NE_Contact(in1 := "dbtags_Sterowanie".HMI.ErrorAck_Int, in2 := 0)
      P_Trig( "dbtags_Sterowanie".HMI.ErrorAck_Int_edge )
      wire#w1
      Coil( "dbtags_Sterowanie".PID_Compact.ErrorAck )
   END_RUNG
   RUNG wire#powerrail
      Contact( "dbtags_Sterowanie".HMI.ErrorAck )
   END_RUNG wire#w1
   RUNG wire#powerrail
      I_Contact( "AlwaysTRUE" )
      { S7_Templates := "SrcType := DWord" } NE_Contact(in1 := "Error_State_PID1", in2 := 0)
      Contact( "InputWarning_L_PID1" )
   END_RUNG wire#w1
   // the same network as SCL:
   #_w1 := "dbtags_Sterowanie".HMI.ErrorAck_Int <> 0;
   #_w2 := #_w1 AND NOT "dbtags_Sterowanie".HMI.ErrorAck_Int_edge;   // rising edge
   "dbtags_Sterowanie".HMI.ErrorAck_Int_edge := #_w1;
   "dbtags_Sterowanie".PID_Compact.ErrorAck := #_w2 OR "dbtags_Sterowanie".HMI.ErrorAck OR (NOT "AlwaysTRUE" AND ("Error_State_PID1" <> 0) AND "InputWarning_L_PID1");
END_REGION
END_ORGANIZATION_BLOCK

ORGANIZATION_BLOCK "Cyclic interrupt_2"   // OB32, LAD, CyclicInterrupt
TITLE = Pobranie analogów z wejścia
{ S7_Optimized_Access := 'TRUE' }
AUTHOR : rtecmer
VERSION : 0.1
// Obsługa wejść analogowych
// stored: AutoNumber true, IsIECCheckEnabled false, SetENOAutomatically false
   VAR_INPUT
      Initial_Call : Bool;   // Initial call of this OB
      Event_Count : Int;   // Events discarded
   END_VAR
BEGIN

REGION Network 1: Pobranie wartości z wejść analogowych
   // B6 - Miasto
   // B7 - Pompownia
   // B8 - Suchobieg
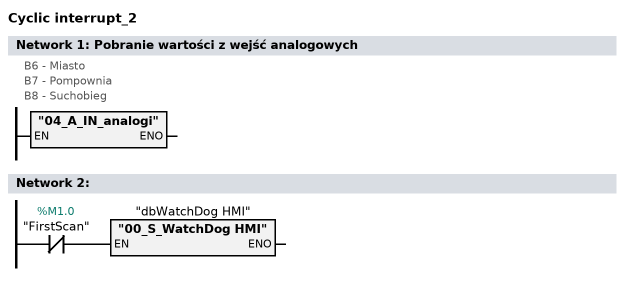
   RUNG wire#powerrail
      "04_A_IN_analogi"()
   END_RUNG
   // the same network as SCL:
   "04_A_IN_analogi"();
END_REGION

REGION Network 2
   RUNG wire#powerrail
      I_Contact( "FirstScan" )
      "dbWatchDog HMI"()
   END_RUNG
   // the same network as SCL:
   IF NOT "FirstScan" THEN
       "dbWatchDog HMI"();   // "00_S_WatchDog HMI"
   END_IF;
END_REGION

REGION Network 3 (SCL): Reset znaczników zbocza wysyłania danych przez TCP
   "memRisingTriger_Data_1" := FALSE;
   "memTrig_Client_Receiving_1" := FALSE;
   "memRisingTriger_Data_2" := FALSE;
   "memTrig_Client_Receiving_2" := FALSE;
   "memRisingTriger_Data_3" := FALSE;
   "memTrig_Client_Receiving_3" := FALSE;
   "memRisingTriger_Data_4" := FALSE;
   "memTrig_Client_Receiving_4" := FALSE;
   "memRisingTriger_Data_5" := FALSE;
   "memTrig_Client_Receiving_5" := FALSE;
   "memRisingTriger_Data_6" := FALSE;
   "memTrig_Client_Receiving_6" := FALSE;
   "memRisingTriger_Data_7" := FALSE;
   "memTrig_Client_Receiving_7" := FALSE;
   "memRisingTriger_Data_8" := FALSE;
   "memTrig_Client_Receiving_8" := FALSE;
   "memRisingTriger_Data_9" := FALSE;
   "memTrig_Client_Receiving_9" := FALSE;
   "memRisingTriger_Data_10" := FALSE;
   "memTrig_Client_Receiving_10" := FALSE;
END_REGION

REGION Network 4 (SCL): pamieć zbocza narastającego przekazania danej do wysłania
   "memRisingTriger_Data_11" := FALSE;
   "memTrig_Client_Receiving_11" := FALSE;
   "memRisingTriger_Data_12" := FALSE;
   "memTrig_Client_Receiving_12" := FALSE;
   "memRisingTriger_Data_13" := FALSE;
   "memTrig_Client_Receiving_13" := FALSE;
   "memRisingTriger_Data_14" := FALSE;
   "memTrig_Client_Receiving_14" := FALSE;
   "memRisingTriger_Data_15" := FALSE;
   "memTrig_Client_Receiving_15" := FALSE;
   "memRisingTriger_Data_16" := FALSE;
   "memTrig_Client_Receiving_16" := FALSE;
   "memRisingTriger_Data_17" := FALSE;
   "memTrig_Client_Receiving_17" := FALSE;
   "memRisingTriger_Data_18" := FALSE;
   "memTrig_Client_Receiving_18" := FALSE;
   "memRisingTriger_Data_19" := FALSE;
   "memTrig_Client_Receiving_19" := FALSE;
   "memRisingTriger_Data_20" := FALSE;
   "memTrig_Client_Receiving_20" := FALSE;
END_REGION
END_ORGANIZATION_BLOCK

FUNCTION "04_A_IN_analogi" : Void
TITLE = Przekazanie wartości z wejść analogowych
{ S7_Optimized_Access := 'TRUE' }
AUTHOR : rtecmer
VERSION : 0.1
//(*
////=============================================================================
////(JZWiK S.A Radosław Tecmer)
////(c)Copyright (2021) All Rights Reserved
////-----------------------------------------------------------------------------
////Testowane z:   (system docelowy z  FW 4.4)
////Pakiet inżynierski:   TIA Portal (V14 Sp1 Update 9)
////Ograniczenia:  ( - )
////Wymagania:  (minimalne S7-1200 CPU 1215C FW 4.2 .)
////Funkcjonalnośc: (Pobranie wartości z wejść analogowych )
////-----------------------------------------------------------------------------
////Zmainy wprowadzone:
////Wersja  Data       Osoba wprowadzająca zmiany - ekspert
////01.00.00 11.01.2022 (Tecmer Radosław - twórca) Pieresza wersja 01.00.00
////=============================================================================
//*)

BEGIN
	(*
	//=============================================================================
	//(JZWiK S.A Radosław Tecmer)
	//(c)Copyright (2021) All Rights Reserved
	//-----------------------------------------------------------------------------
	//Testowane z:   (system docelowy z  FW 4.4)
	//Pakiet inżynierski:   TIA Portal (V14 Sp1 Update 9)
	//Ograniczenia:  ( - )
	//Wymagania:  (minimalne S7-1200 CPU 1215C FW 4.2 .)
	//Funkcjonalnośc: (Pobranie wartości z wejść analogowych )
	//-----------------------------------------------------------------------------
	//Zmainy wprowadzone:
	//Wersja  Data       Osoba wprowadzająca zmiany - ekspert
	//01.00.00 11.01.2022 (Tecmer Radosław - twórca) Pieresza wersja 01.00.00
	//=============================================================================
	*)
	
	// ciśnienie przetłaczania straefa 2
	IF "dbdane".PV_analaog_B6 > 0.2 THEN // czy nie uszkodzone rury
	  IF "dbdane".PV_analaog_B6 < 27651 THEN // przerwana pętla prądowa
	    // to przekazanie wartości
	    "dbdane".PV_PER_B6 := "dbdane".PV_analaog_B6;
	  ELSE
	    "dbdane".PV_PER_B6 := 32767;
	    ;
	  END_IF;
	  
	  ;
	END_IF;
	
	
	
	// ciśnienie strefa 1
	IF "dbdane".PV_analaog_B7 > 0.2 THEN // czy nie uszkodzone rury
	  IF "dbdane".PV_analaog_B7 < 27651 THEN // przerwana pętla prądowa
	    // to przekazanie wartości
	    "dbdane".PV_PER_B5 := "dbdane".PV_analaog_B7;
	    ;
	  ELSE
	    "dbdane".PV_PER_B5 := 32767;
	    ;
	  END_IF;
	  
	  ;
	END_IF;
	
	
	//ciśnienie ssania
	IF  "dbdane".PV_analaog_B8 > 0.2 THEN // czy nie uszkodzone rury
	  // to przekazanie wartości
	  "dbdane".PV_PER_B8 := "dbdane".PV_analaog_B8;
	ELSE
	  "dbdane".PV_PER_B8 := 0;
	  ;
	END_IF;
	
	
	REGION Zbiornik duży 3
	  //Kontrola stanu pomiaru 
	  IF "dbdane".actSignalTank3 >= 0.2 THEN
	    // przekaż do skady 
	    "dbdane".actLevel_Tank3 := "dbdane".actValu_Tank3;
	  ELSE
	    "dbdane".actLevel_Tank3 := 400; // jeśli alarm to ustaw 400cm
	    
	    ;
	  END_IF;
	  
	  
	  
	END_REGION
	
	REGION Zbiorniki małe  1
	  //Kontrola stanu pomiaru 
	  IF "dbdane".actSignalTank1 >= 0.2 THEN
	    // przekaż do skady 
	    "dbdane".actLevel_Tank1 := "dbdane".actValu_Tank1;
	  ELSE
	    "dbdane".actLevel_Tank1 := 400; // jeśli alarm to ustaw 400cm
	    
	    ;
	  END_IF;
	  
	  
	  
	END_REGION
	
	REGION Zbiorniki małe  2
	  //Kontrola stanu pomiaru 
	  IF "dbdane".actSignalTank2 >= 0.2 THEN
	    // przekaż do skady 
	    "dbdane".actLevel_Tank2 := "dbdane".actValu_Tank2;
	  ELSE
	    "dbdane".actLevel_Tank2 := 400; // jeśli alarm to ustaw 400cm
	    
	    ;
	  END_IF;
	  
	  
	  
	END_REGION
	
	// --------!!!!!!!!!!!   Do opracowania czy pomiar będzie z impulsów czy ModbusRTU
	// przepływ analog
	//"dbdane".actPrzepływQ1_IA := 27648;
	
	//"dbdane".actPrzepływQ1_IA_real := "00_S_SclScaleLinearIntToReal"(x := "dbdane".actPrzepływQ1_IA, yMin := 0.0, yMax := 600.0, y0 := 0.0, x0 := 0, x1 := 27648, y1 := 600.0);
	
END_FUNCTION

FUNCTION_BLOCK "00_S_WatchDog HMI"   // FB12, LAD
TITLE = WatchDog HMI
{ S7_Optimized_Access := 'TRUE' }
AUTHOR : rtecmer
VERSION : 0.1
// Kontrola komunikacji PLC z HMI.  Wartość w zmiennej w instancji "Dane_ComunicationControlHMI".tempCoordinationHMIRS5 jest inkrementowana przez PLC i co minutę skrypt z HMI wartość zeruje. Jeśli błąd kumunikacj to wartość jest inkrementowana do max zmiennej. Przy wartości 70 ustawiany jest bit alarmu dla PLC, że btrak komunikacji z HMI
// HMI na podstawie błędu systemowego 190011 komonikuje w tabeli alarmów o braku komunikacji
// stored: AutoNumber true, IsIECCheckEnabled false, IsRetainMemResEnabled false, MemoryReserve 500, SetENOAutomatically false, UDAEnableTagReadback false
   VAR_TEMP   // added for the SCL form of the ladder/FBD networks
      _w1 : Bool;
      _w2 : Bool;
   END_VAR
BEGIN

REGION Network 1: WatchDog HMI
   // Do zrobienia
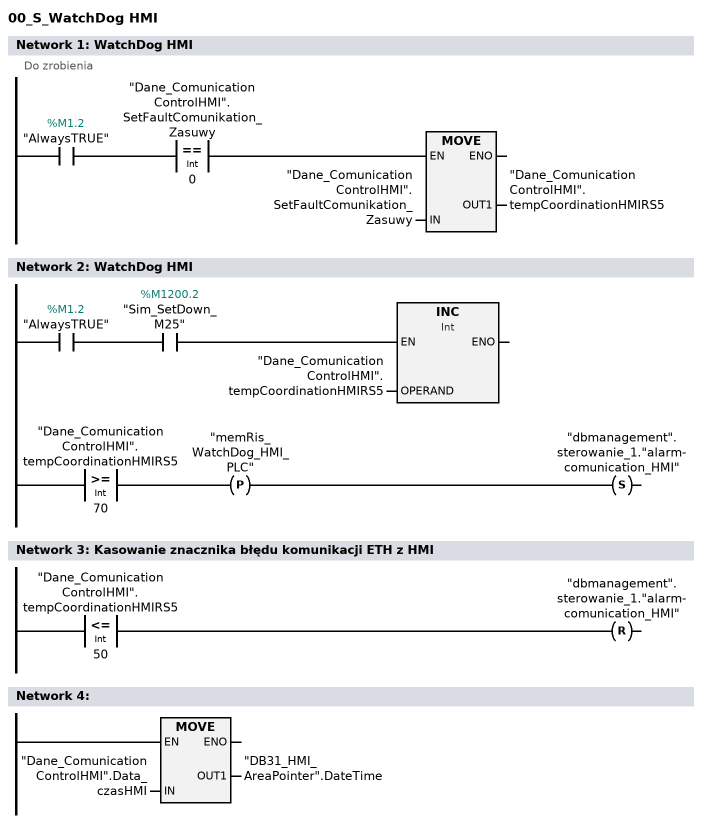
   RUNG wire#powerrail
      Contact( "AlwaysTRUE" )
      { S7_Templates := "SrcType := Int" } EQ_Contact(in1 := "Dane_ComunicationControlHMI".SetFaultComunikation_Zasuwy, in2 := 0)
      Move(in := "Dane_ComunicationControlHMI".SetFaultComunikation_Zasuwy, out1 => "Dane_ComunicationControlHMI".tempCoordinationHMIRS5)
   END_RUNG
   // the same network as SCL:
   IF "AlwaysTRUE" AND ("Dane_ComunicationControlHMI".SetFaultComunikation_Zasuwy = 0) THEN
       "Dane_ComunicationControlHMI".tempCoordinationHMIRS5 := "Dane_ComunicationControlHMI".SetFaultComunikation_Zasuwy;
   END_IF;
END_REGION

REGION Network 2: WatchDog HMI
   RUNG wire#powerrail
      Contact( "AlwaysTRUE" )
      Contact( "Sim_SetDown_M25" )
      { S7_Templates := "DestType := Int" } Inc( "Dane_ComunicationControlHMI".tempCoordinationHMIRS5 )
   END_RUNG
   RUNG wire#powerrail
      { S7_Templates := "SrcType := Int" } GE_Contact(in1 := "Dane_ComunicationControlHMI".tempCoordinationHMIRS5, in2 := 70)
      P_Trig( "memRis_WatchDog_HMI_PLC" )
      S_Coil( "dbmanagement".sterowanie_1."alarm-comunication_HMI" )
   END_RUNG
   // the same network as SCL:
   IF "AlwaysTRUE" AND "Sim_SetDown_M25" THEN
       "Dane_ComunicationControlHMI".tempCoordinationHMIRS5 := "Dane_ComunicationControlHMI".tempCoordinationHMIRS5 + 1;
   END_IF;
   #_w1 := "Dane_ComunicationControlHMI".tempCoordinationHMIRS5 >= 70;
   #_w2 := #_w1 AND NOT "memRis_WatchDog_HMI_PLC";   // rising edge
   "memRis_WatchDog_HMI_PLC" := #_w1;
   IF #_w2 THEN "dbmanagement".sterowanie_1."alarm-comunication_HMI" := TRUE; END_IF;
END_REGION

REGION Network 3: Kasowanie znacznika błędu komunikacji ETH z HMI
   RUNG wire#powerrail
      { S7_Templates := "SrcType := Int" } LE_Contact(in1 := "Dane_ComunicationControlHMI".tempCoordinationHMIRS5, in2 := 50)
      R_Coil( "dbmanagement".sterowanie_1."alarm-comunication_HMI" )
   END_RUNG
   // the same network as SCL:
   IF "Dane_ComunicationControlHMI".tempCoordinationHMIRS5 <= 50 THEN
       "dbmanagement".sterowanie_1."alarm-comunication_HMI" := FALSE;
   END_IF;
END_REGION

REGION Network 4
   RUNG wire#powerrail
      Move(in := "Dane_ComunicationControlHMI".Data_czasHMI, out1 => "DB31_HMI_AreaPointer".DateTime)
   END_RUNG
   // the same network as SCL:
   "DB31_HMI_AreaPointer".DateTime := "Dane_ComunicationControlHMI".Data_czasHMI;
END_REGION
END_FUNCTION_BLOCK

ORGANIZATION_BLOCK "Cyclic interrupt_SlaveModbusRTU"   // OB31, LAD, CyclicInterrupt
{ S7_Optimized_Access := 'TRUE' }
AUTHOR : rtecmer
VERSION : 0.1
// stored: AutoNumber true, IsIECCheckEnabled false, SetENOAutomatically false
   VAR_INPUT
      Initial_Call : Bool;   // Initial call of this OB
      Event_Count : Int;   // Events discarded
   END_VAR
BEGIN

REGION Network 1
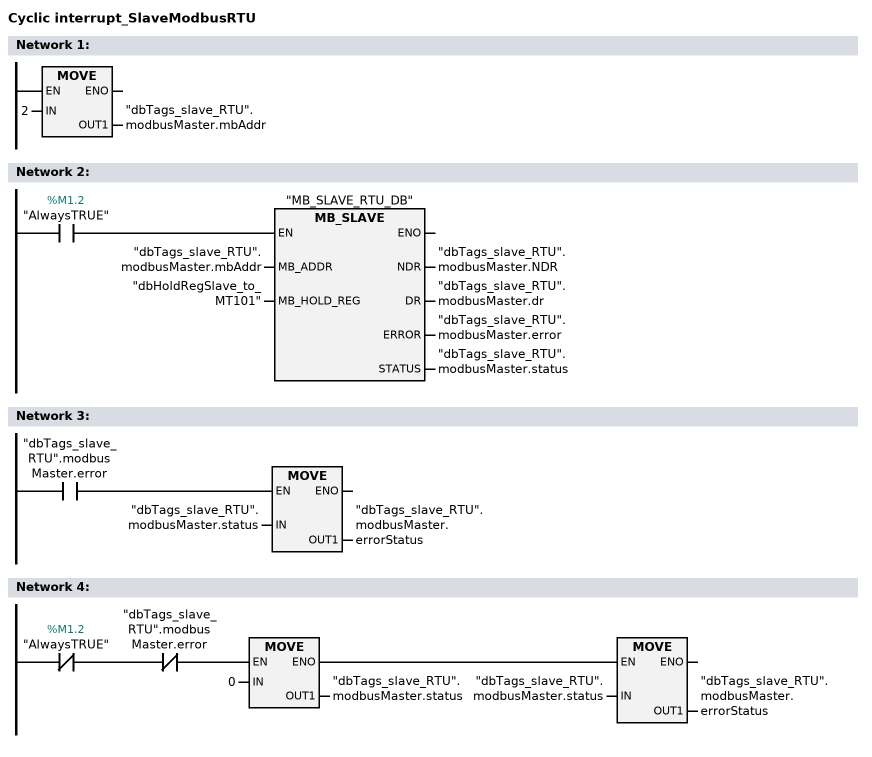
   RUNG wire#powerrail
      Move(in := 2, out1 => "dbTags_slave_RTU".modbusMaster.mbAddr)
   END_RUNG
   // the same network as SCL:
   "dbTags_slave_RTU".modbusMaster.mbAddr := 2;
END_REGION

REGION Network 2
   RUNG wire#powerrail
      Contact( "AlwaysTRUE" )
      "MB_SLAVE_RTU_DB".MB_SLAVE(MB_ADDR := "dbTags_slave_RTU".modbusMaster.mbAddr, MB_HOLD_REG := "dbHoldRegSlave_to_MT101", NDR => "dbTags_slave_RTU".modbusMaster.NDR, DR => "dbTags_slave_RTU".modbusMaster.dr, ERROR => "dbTags_slave_RTU".modbusMaster.error, STATUS => "dbTags_slave_RTU".modbusMaster.status)
   END_RUNG
   // the same network as SCL:
   IF "AlwaysTRUE" THEN
       "MB_SLAVE_RTU_DB"(MB_ADDR := "dbTags_slave_RTU".modbusMaster.mbAddr,   // MB_SLAVE
                         MB_HOLD_REG := "dbHoldRegSlave_to_MT101",
                         NDR => "dbTags_slave_RTU".modbusMaster.NDR,
                         DR => "dbTags_slave_RTU".modbusMaster.dr,
                         ERROR => "dbTags_slave_RTU".modbusMaster.error,
                         STATUS => "dbTags_slave_RTU".modbusMaster.status);
   END_IF;
END_REGION

REGION Network 3
   RUNG wire#powerrail
      Contact( "dbTags_slave_RTU".modbusMaster.error )
      Move(in := "dbTags_slave_RTU".modbusMaster.status, out1 => "dbTags_slave_RTU".modbusMaster.errorStatus)
   END_RUNG
   // the same network as SCL:
   IF "dbTags_slave_RTU".modbusMaster.error THEN
       "dbTags_slave_RTU".modbusMaster.errorStatus := "dbTags_slave_RTU".modbusMaster.status;
   END_IF;
END_REGION

REGION Network 4
   RUNG wire#powerrail
      I_Contact( "AlwaysTRUE" )
      I_Contact( "dbTags_slave_RTU".modbusMaster.error )
      Move(in := 0, out1 => "dbTags_slave_RTU".modbusMaster.status)
      Move(in := "dbTags_slave_RTU".modbusMaster.status, out1 => "dbTags_slave_RTU".modbusMaster.errorStatus)
   END_RUNG
   // the same network as SCL:
   IF NOT "AlwaysTRUE" AND NOT "dbTags_slave_RTU".modbusMaster.error THEN
       "dbTags_slave_RTU".modbusMaster.status := 0;
       "dbTags_slave_RTU".modbusMaster.errorStatus := "dbTags_slave_RTU".modbusMaster.status;
   END_IF;
END_REGION
END_ORGANIZATION_BLOCK

ORGANIZATION_BLOCK "Diagnostic error interrupt"   // OB82, LAD, DiagnosticErrorInterrupt
TITLE = Diagnostyka błedów
{ S7_Optimized_Access := 'TRUE' }
AUTHOR : rtecmer
VERSION : 0.1
// stored: IsIECCheckEnabled false, SetENOAutomatically false
   VAR_INPUT
      IO_State : Word;   // IO state of the HW object
      LADDR : HW_ANY;   // Hardware identifier
      Channel : UInt;   // Channel number
      MultiError : Bool;   // =true if more than one error is present
   END_VAR
   VAR_TEMP
      RetVal_RD_SYS_T : Int;   // //Status of the instruction RD_SYS_T: Read time-of-day
   END_VAR
BEGIN

REGION Network 2 (SCL)
   "EX012_ErrorBuffer_OB82".OB82ErrorCounter := "EX012_ErrorBuffer_OB82".OB82ErrorCounter + 1;
   //ochrona przed przepełnieniem tabeli
   IF ("EX012_ErrorBuffer_OB82".OB82ErrorCounter > "CONST_BUFFER_OB82") THEN
     "EX012_ErrorBuffer_OB82".OB82ErrorCounter := 1;
   END_IF;
   //Wystąpił błąd czasu
   #RetVal_RD_SYS_T := RD_LOC_T(OUT => "EX012_ErrorBuffer_OB82".ErrorDataOB82["EX012_ErrorBuffer_OB82".OB82ErrorCounter].ErrorTimestamp);
   //Zapis błedu do buffora (ErrorBuffor)
   "EX012_ErrorBuffer_OB82".ErrorDataOB82["EX012_ErrorBuffer_OB82".OB82ErrorCounter].IO_State := #IO_State;
   "EX012_ErrorBuffer_OB82".ErrorDataOB82["EX012_ErrorBuffer_OB82".OB82ErrorCounter].LADDR := #LADDR;
   "EX012_ErrorBuffer_OB82".ErrorDataOB82["EX012_ErrorBuffer_OB82".OB82ErrorCounter].Channel := #Channel;
   "EX012_ErrorBuffer_OB82".ErrorDataOB82["EX012_ErrorBuffer_OB82".OB82ErrorCounter].MultiError := #MultiError;
END_REGION
END_ORGANIZATION_BLOCK

ORGANIZATION_BLOCK "Hardware interrupt Reset"   // OB40, LAD, HardwareInterrupt
TITLE = Reset
{ S7_Optimized_Access := 'TRUE' }
AUTHOR : rtecmer
VERSION : 0.1
// Ustawienie gotowości i tryb
// stored: AutoNumber true, IsIECCheckEnabled false, SetENOAutomatically false
   VAR_INPUT
      LADDR : HW_IO;   // Hardware identifier
      USI : Word;   // User structure identifier
      IChannel : USInt;   // Interrupt channel number
      EventType : Byte;   // EventType
   END_VAR
BEGIN
END_ORGANIZATION_BLOCK

ORGANIZATION_BLOCK "Reset_falling_edge_PowerRS5"   // OB41, LAD, HardwareInterrupt
TITLE = Reset po braku zasilania RS5
{ S7_Optimized_Access := 'TRUE' }
AUTHOR : rtecmer
VERSION : 0.1
// Reset napędów po braku zasilania przy opadającym zboczu Power RS5
// stored: AutoNumber true, IsIECCheckEnabled false, SetENOAutomatically false
   VAR_INPUT
      LADDR : HW_IO;   // Hardware identifier
      USI : Word;   // User structure identifier
      IChannel : USInt;   // Interrupt channel number
      EventType : Byte;   // EventType
   END_VAR
BEGIN
END_ORGANIZATION_BLOCK

ORGANIZATION_BLOCK "Startup"   // OB100, LAD, Startup
TITLE = "Complete Restart"
{ S7_Optimized_Access := 'TRUE' }
AUTHOR : RTecmer
VERSION : 0.1
// stored: AutoNumber true, IsIECCheckEnabled false, SetENOAutomatically false
   VAR_INPUT
      LostRetentive : Bool;   // True if retentive data are lost
      LostRTC : Bool;   // True if date and time are lost
   END_VAR
BEGIN

REGION Network 1: inicjacja master modbus RTU / Incjalizacja modułu Master CM1241 (RS485) Modbus RTU
   // Komunikacja z przepływomierzami ABB i falownikiem Danfoss
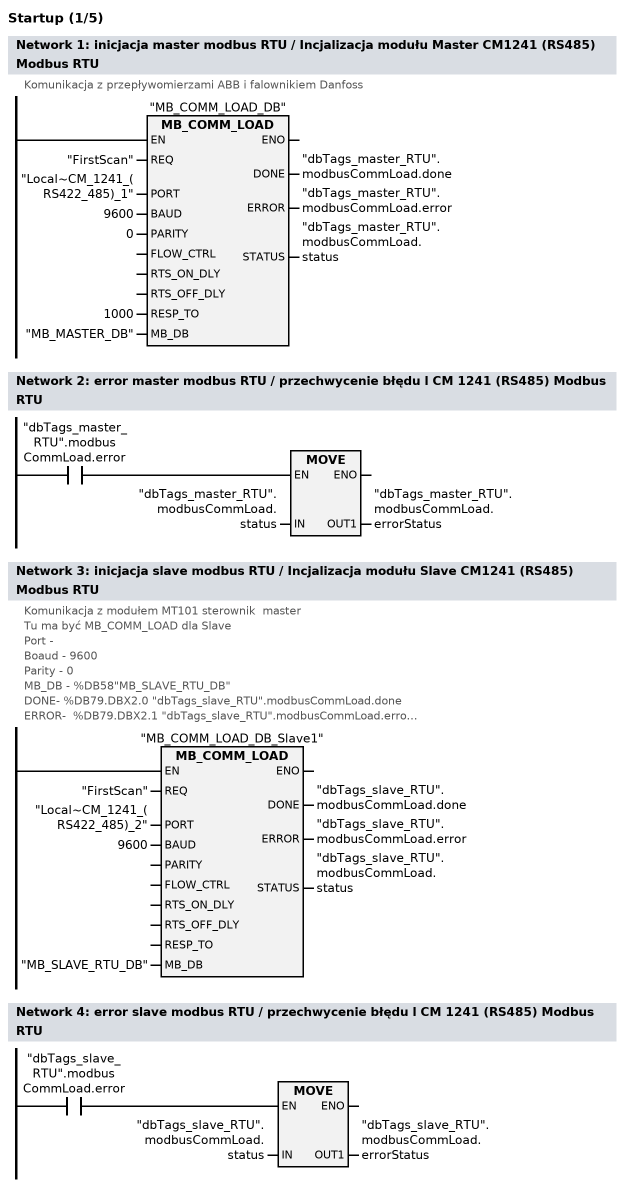
   RUNG wire#powerrail
      "MB_COMM_LOAD_DB".MB_COMM_LOAD(REQ := "FirstScan", PORT := "Local~CM_1241_(RS422_485)_1", BAUD := 9600, PARITY := 0, FLOW_CTRL :=, RTS_ON_DLY :=, RTS_OFF_DLY :=, RESP_TO := 1000, MB_DB := "MB_MASTER_DB", DONE => "dbTags_master_RTU".modbusCommLoad.done, ERROR => "dbTags_master_RTU".modbusCommLoad.error, STATUS => "dbTags_master_RTU".modbusCommLoad.status)
   END_RUNG
   // the same network as SCL:
   "MB_COMM_LOAD_DB"(REQ := "FirstScan",   // MB_COMM_LOAD
                     PORT := "Local~CM_1241_(RS422_485)_1",
                     BAUD := 9600,
                     PARITY := 0,
                     RESP_TO := 1000,
                     MB_DB := "MB_MASTER_DB",
                     DONE => "dbTags_master_RTU".modbusCommLoad.done,
                     ERROR => "dbTags_master_RTU".modbusCommLoad.error,
                     STATUS => "dbTags_master_RTU".modbusCommLoad.status);
END_REGION

REGION Network 2: error master modbus RTU / przechwycenie błędu l CM 1241 (RS485) Modbus RTU
   RUNG wire#powerrail
      Contact( "dbTags_master_RTU".modbusCommLoad.error )
      { S7_GenerateENO := "TRUE" } Move(in := "dbTags_master_RTU".modbusCommLoad.status, out1 => "dbTags_master_RTU".modbusCommLoad.errorStatus)
   END_RUNG
   // the same network as SCL:
   IF "dbTags_master_RTU".modbusCommLoad.error THEN
       "dbTags_master_RTU".modbusCommLoad.errorStatus := "dbTags_master_RTU".modbusCommLoad.status;
   END_IF;
END_REGION

REGION Network 3: inicjacja slave modbus RTU / Incjalizacja modułu Slave CM1241 (RS485) Modbus RTU
   // Komunikacja z modułem MT101 sterownik  master
   // 
   // Tu ma być MB_COMM_LOAD dla Slave
   // Port -
   // Boaud - 9600
   // Parity - 0
   // MB_DB - %DB58"MB_SLAVE_RTU_DB"
   // DONE- %DB79.DBX2.0 "dbTags_slave_RTU".modbusCommLoad.done
   // ERROR-  %DB79.DBX2.1 "dbTags_slave_RTU".modbusCommLoad.error
   // STATUS - %DB79.DBX2.2 "dbTags_slave_RTU".modbusCommLoad.status
   RUNG wire#powerrail
      "MB_COMM_LOAD_DB_Slave1".MB_COMM_LOAD(REQ := "FirstScan", PORT := "Local~CM_1241_(RS422_485)_2", BAUD := 9600, PARITY :=, FLOW_CTRL :=, RTS_ON_DLY :=, RTS_OFF_DLY :=, RESP_TO :=, MB_DB := "MB_SLAVE_RTU_DB", DONE => "dbTags_slave_RTU".modbusCommLoad.done, ERROR => "dbTags_slave_RTU".modbusCommLoad.error, STATUS => "dbTags_slave_RTU".modbusCommLoad.status)
   END_RUNG
   // the same network as SCL:
   "MB_COMM_LOAD_DB_Slave1"(REQ := "FirstScan",   // MB_COMM_LOAD
                           PORT := "Local~CM_1241_(RS422_485)_2",
                           BAUD := 9600,
                           MB_DB := "MB_SLAVE_RTU_DB",
                           DONE => "dbTags_slave_RTU".modbusCommLoad.done,
                           ERROR => "dbTags_slave_RTU".modbusCommLoad.error,
                           STATUS => "dbTags_slave_RTU".modbusCommLoad.status);
END_REGION

REGION Network 4: error slave modbus RTU / przechwycenie błędu l CM 1241 (RS485) Modbus RTU
   RUNG wire#powerrail
      Contact( "dbTags_slave_RTU".modbusCommLoad.error )
      { S7_GenerateENO := "TRUE" } Move(in := "dbTags_slave_RTU".modbusCommLoad.status, out1 => "dbTags_slave_RTU".modbusCommLoad.errorStatus)
   END_RUNG
   // the same network as SCL:
   IF "dbTags_slave_RTU".modbusCommLoad.error THEN
       "dbTags_slave_RTU".modbusCommLoad.errorStatus := "dbTags_slave_RTU".modbusCommLoad.status;
   END_IF;
END_REGION

REGION Network 5: Znacznik dodatkowej pompy dla funkcji FB8 I / Znacznik dodatkowego kompresora dla funkcji FB8 I
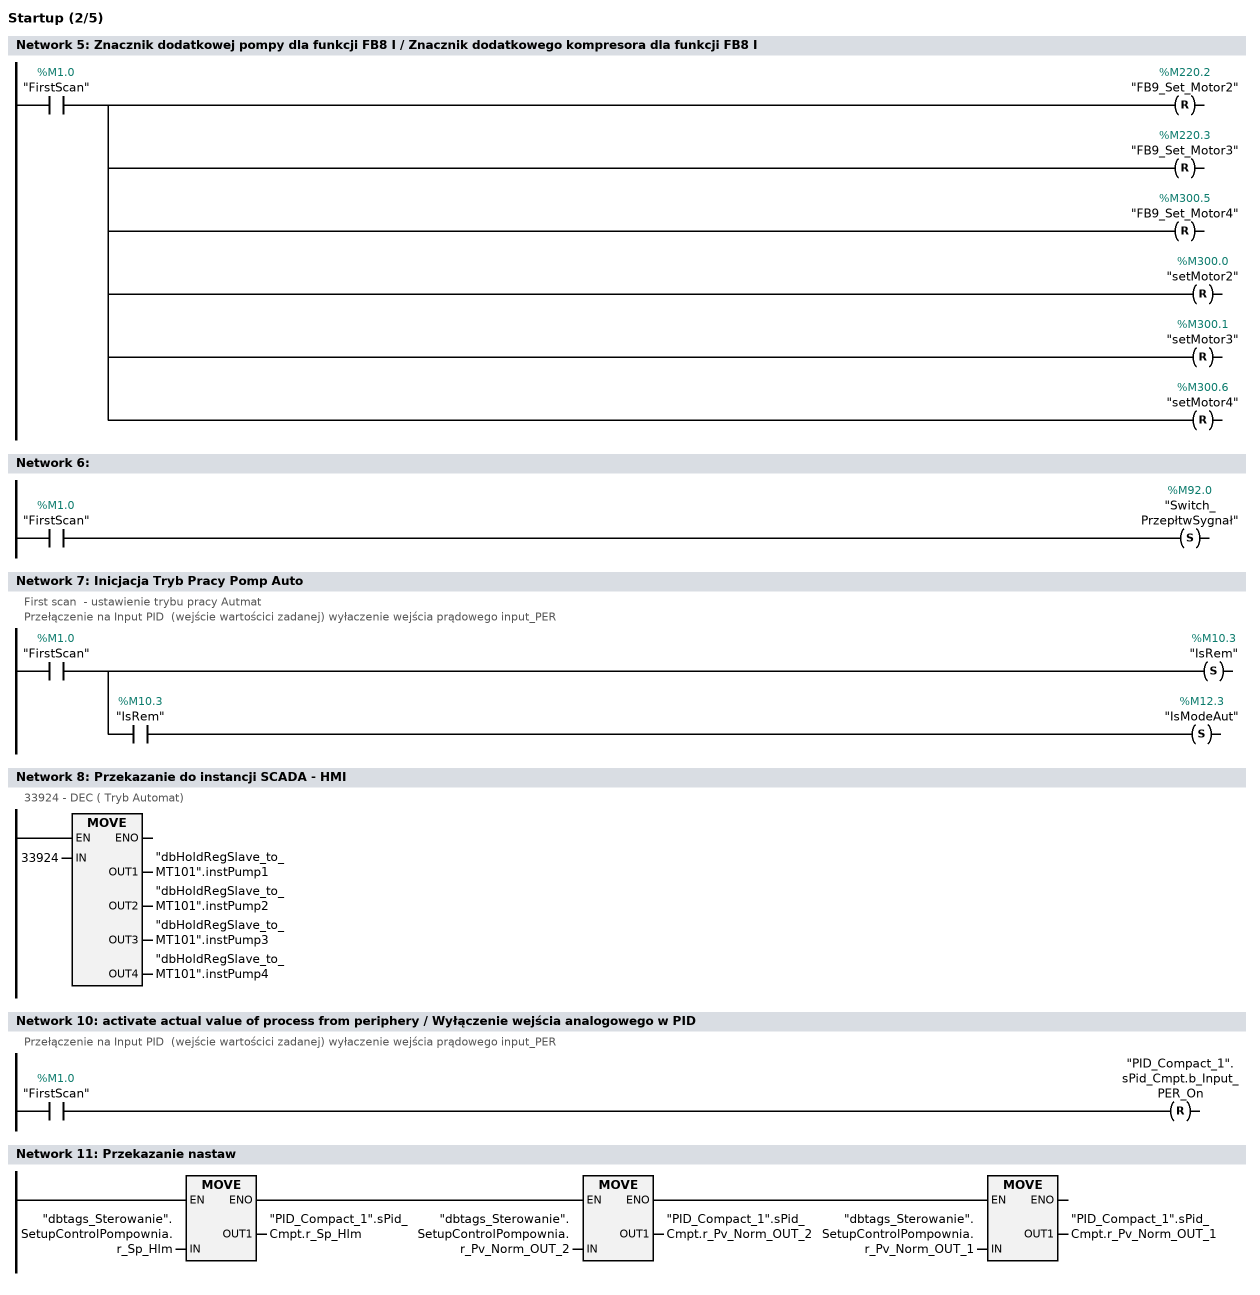
   RUNG wire#powerrail
      Contact( "FirstScan" )
      wire#w1
      R_Coil( "FB9_Set_Motor2" )
   END_RUNG
   RUNG wire#w1
      R_Coil( "FB9_Set_Motor3" )
   END_RUNG
   RUNG wire#w1
      R_Coil( "FB9_Set_Motor4" )
   END_RUNG
   RUNG wire#w1
      R_Coil( "setMotor2" )
   END_RUNG
   RUNG wire#w1
      R_Coil( "setMotor3" )
   END_RUNG
   RUNG wire#w1
      R_Coil( "setMotor4" )
   END_RUNG
   // the same network as SCL:
   IF "FirstScan" THEN
       "FB9_Set_Motor2" := FALSE;
       "FB9_Set_Motor3" := FALSE;
       "FB9_Set_Motor4" := FALSE;
       "setMotor2" := FALSE;
       "setMotor3" := FALSE;
       "setMotor4" := FALSE;
   END_IF;
END_REGION

REGION Network 6
   RUNG wire#powerrail
      Contact( "FirstScan" )
      S_Coil( "Switch_PrzepłtwSygnał" )
   END_RUNG
   // the same network as SCL:
   IF "FirstScan" THEN "Switch_PrzepłtwSygnał" := TRUE; END_IF;
END_REGION

REGION Network 7: Inicjacja Tryb Pracy Pomp Auto
   // First scan  - ustawienie trybu pracy Autmat 
   // Przełączenie na Input PID  (wejście wartościci zadanej) wyłaczenie wejścia prądowego input_PER
   RUNG wire#powerrail
      Contact( "FirstScan" )
      wire#w1
      S_Coil( "IsRem" )
   END_RUNG
   RUNG wire#w1
      Contact( "IsRem" )
      S_Coil( "IsModeAut" )
   END_RUNG
   // the same network as SCL:
   IF "FirstScan" THEN "IsRem" := TRUE; END_IF;
   IF "FirstScan" AND "IsRem" THEN "IsModeAut" := TRUE; END_IF;
END_REGION

REGION Network 8: Przekazanie do instancji SCADA - HMI
   // 33924 - DEC ( Tryb Automat)
   RUNG wire#powerrail
      { S7_GenerateENO := "TRUE" } Move(in := 33924, out1 => "dbHoldRegSlave_to_MT101".instPump1, out2 => "dbHoldRegSlave_to_MT101".instPump2, out3 => "dbHoldRegSlave_to_MT101".instPump3, out4 => "dbHoldRegSlave_to_MT101".instPump4)
   END_RUNG
   // the same network as SCL:
   "dbHoldRegSlave_to_MT101".instPump1 := 33924;
   "dbHoldRegSlave_to_MT101".instPump2 := 33924;
   "dbHoldRegSlave_to_MT101".instPump3 := 33924;
   "dbHoldRegSlave_to_MT101".instPump4 := 33924;
END_REGION

REGION Network 10: activate actual value of process from periphery / Wyłączenie wejścia analogowego w PID
   // Przełączenie na Input PID  (wejście wartościci zadanej) wyłaczenie wejścia prądowego input_PER
   RUNG wire#powerrail
      Contact( "FirstScan" )
      R_Coil( "PID_Compact_1".sPid_Cmpt.b_Input_PER_On )
   END_RUNG
   // the same network as SCL:
   IF "FirstScan" THEN "PID_Compact_1".sPid_Cmpt.b_Input_PER_On := FALSE; END_IF;
END_REGION

REGION Network 11: Przekazanie nastaw
   RUNG wire#powerrail
      { S7_GenerateENO := "TRUE" } Move(in := "dbtags_Sterowanie".SetupControlPompownia.r_Sp_Hlm, out1 => "PID_Compact_1".sPid_Cmpt.r_Sp_Hlm)
      { S7_GenerateENO := "TRUE" } Move(in := "dbtags_Sterowanie".SetupControlPompownia.r_Pv_Norm_OUT_2, out1 => "PID_Compact_1".sPid_Cmpt.r_Pv_Norm_OUT_2)
      { S7_GenerateENO := "TRUE" } Move(in := "dbtags_Sterowanie".SetupControlPompownia.r_Pv_Norm_OUT_1, out1 => "PID_Compact_1".sPid_Cmpt.r_Pv_Norm_OUT_1)
   END_RUNG
   // the same network as SCL:
   // ENO of a box is taken as its EN; it also drops when the box reports an error
   "PID_Compact_1".sPid_Cmpt.r_Sp_Hlm := "dbtags_Sterowanie".SetupControlPompownia.r_Sp_Hlm;
   "PID_Compact_1".sPid_Cmpt.r_Pv_Norm_OUT_2 := "dbtags_Sterowanie".SetupControlPompownia.r_Pv_Norm_OUT_2;
   "PID_Compact_1".sPid_Cmpt.r_Pv_Norm_OUT_1 := "dbtags_Sterowanie".SetupControlPompownia.r_Pv_Norm_OUT_1;
END_REGION

REGION Network 12: Inicjacja nastaw PID
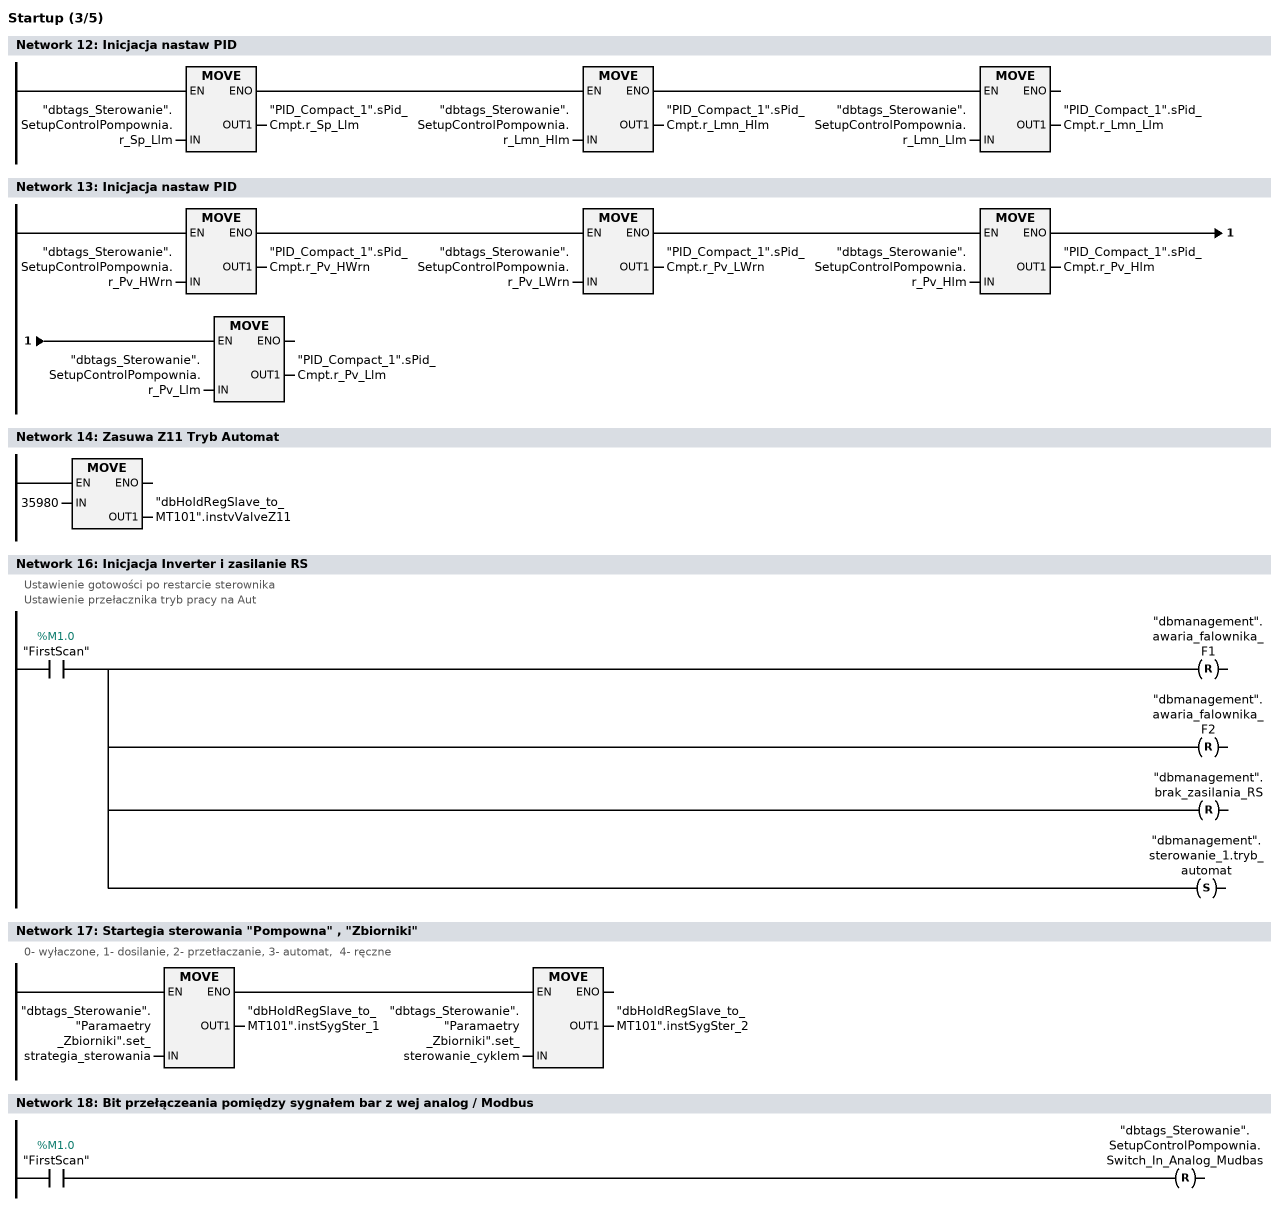
   RUNG wire#powerrail
      { S7_GenerateENO := "TRUE" } Move(in := "dbtags_Sterowanie".SetupControlPompownia.r_Sp_Llm, out1 => "PID_Compact_1".sPid_Cmpt.r_Sp_Llm)
      { S7_GenerateENO := "TRUE" } Move(in := "dbtags_Sterowanie".SetupControlPompownia.r_Lmn_Hlm, out1 => "PID_Compact_1".sPid_Cmpt.r_Lmn_Hlm)
      { S7_GenerateENO := "TRUE" } Move(in := "dbtags_Sterowanie".SetupControlPompownia.r_Lmn_Llm, out1 => "PID_Compact_1".sPid_Cmpt.r_Lmn_Llm)
   END_RUNG
   // the same network as SCL:
   // ENO of a box is taken as its EN; it also drops when the box reports an error
   "PID_Compact_1".sPid_Cmpt.r_Sp_Llm := "dbtags_Sterowanie".SetupControlPompownia.r_Sp_Llm;
   "PID_Compact_1".sPid_Cmpt.r_Lmn_Hlm := "dbtags_Sterowanie".SetupControlPompownia.r_Lmn_Hlm;
   "PID_Compact_1".sPid_Cmpt.r_Lmn_Llm := "dbtags_Sterowanie".SetupControlPompownia.r_Lmn_Llm;
END_REGION

REGION Network 13: Inicjacja nastaw PID
   RUNG wire#powerrail
      { S7_GenerateENO := "TRUE" } Move(in := "dbtags_Sterowanie".SetupControlPompownia.r_Pv_HWrn, out1 => "PID_Compact_1".sPid_Cmpt.r_Pv_HWrn)
      { S7_GenerateENO := "TRUE" } Move(in := "dbtags_Sterowanie".SetupControlPompownia.r_Pv_LWrn, out1 => "PID_Compact_1".sPid_Cmpt.r_Pv_LWrn)
      { S7_GenerateENO := "TRUE" } Move(in := "dbtags_Sterowanie".SetupControlPompownia.r_Pv_Hlm, out1 => "PID_Compact_1".sPid_Cmpt.r_Pv_Hlm)
      { S7_GenerateENO := "TRUE" } Move(in := "dbtags_Sterowanie".SetupControlPompownia.r_Pv_Llm, out1 => "PID_Compact_1".sPid_Cmpt.r_Pv_Llm)
   END_RUNG
   // the same network as SCL:
   // ENO of a box is taken as its EN; it also drops when the box reports an error
   "PID_Compact_1".sPid_Cmpt.r_Pv_HWrn := "dbtags_Sterowanie".SetupControlPompownia.r_Pv_HWrn;
   "PID_Compact_1".sPid_Cmpt.r_Pv_LWrn := "dbtags_Sterowanie".SetupControlPompownia.r_Pv_LWrn;
   "PID_Compact_1".sPid_Cmpt.r_Pv_Hlm := "dbtags_Sterowanie".SetupControlPompownia.r_Pv_Hlm;
   "PID_Compact_1".sPid_Cmpt.r_Pv_Llm := "dbtags_Sterowanie".SetupControlPompownia.r_Pv_Llm;
END_REGION

REGION Network 14: Zasuwa Z11 Tryb Automat
   RUNG wire#powerrail
      Move(in := 35980, out1 => "dbHoldRegSlave_to_MT101".instvValveZ11)
   END_RUNG
   // the same network as SCL:
   "dbHoldRegSlave_to_MT101".instvValveZ11 := 35980;
END_REGION

REGION Network 16: Inicjacja Inverter i zasilanie RS
   // Ustawienie gotowości po restarcie sterownika
   // Ustawienie przełacznika tryb pracy na Aut
   RUNG wire#powerrail
      Contact( "FirstScan" )
      wire#w1
      R_Coil( "dbmanagement".awaria_falownika_F1 )
   END_RUNG
   RUNG wire#w1
      R_Coil( "dbmanagement".awaria_falownika_F2 )
   END_RUNG
   RUNG wire#w1
      R_Coil( "dbmanagement".brak_zasilania_RS )
   END_RUNG
   RUNG wire#w1
      S_Coil( "dbmanagement".sterowanie_1.tryb_automat )
   END_RUNG
   // the same network as SCL:
   IF "FirstScan" THEN
       "dbmanagement".awaria_falownika_F1 := FALSE;
       "dbmanagement".awaria_falownika_F2 := FALSE;
       "dbmanagement".brak_zasilania_RS := FALSE;
       "dbmanagement".sterowanie_1.tryb_automat := TRUE;
   END_IF;
END_REGION

REGION Network 17: Startegia sterowania "Pompowna" , "Zbiorniki"
   // 0- wyłaczone, 1- dosilanie, 2- przetłaczanie, 3- automat,  4- ręczne
   RUNG wire#powerrail
      Move(in := "dbtags_Sterowanie"."Paramaetry _Zbiorniki".set_strategia_sterowania, out1 => "dbHoldRegSlave_to_MT101".instSygSter_1)
      Move(in := "dbtags_Sterowanie"."Paramaetry _Zbiorniki".set_sterowanie_cyklem, out1 => "dbHoldRegSlave_to_MT101".instSygSter_2)
   END_RUNG
   // the same network as SCL:
   "dbHoldRegSlave_to_MT101".instSygSter_1 := "dbtags_Sterowanie"."Paramaetry _Zbiorniki".set_strategia_sterowania;
   "dbHoldRegSlave_to_MT101".instSygSter_2 := "dbtags_Sterowanie"."Paramaetry _Zbiorniki".set_sterowanie_cyklem;
END_REGION

REGION Network 18: Bit przełączeania pomiędzy sygnałem bar z wej analog / Modbus
   RUNG wire#powerrail
      Contact( "FirstScan" )
      R_Coil( "dbtags_Sterowanie".SetupControlPompownia.Switch_In_Analog_Mudbas )
   END_RUNG
   // the same network as SCL:
   IF "FirstScan" THEN "dbtags_Sterowanie".SetupControlPompownia.Switch_In_Analog_Mudbas := FALSE; END_IF;
END_REGION

REGION Network 19: Inicjacja modbus rtu / Modbus RTU start
   // Uwaga !!: Tylko jedna pętla może być uruchomiona
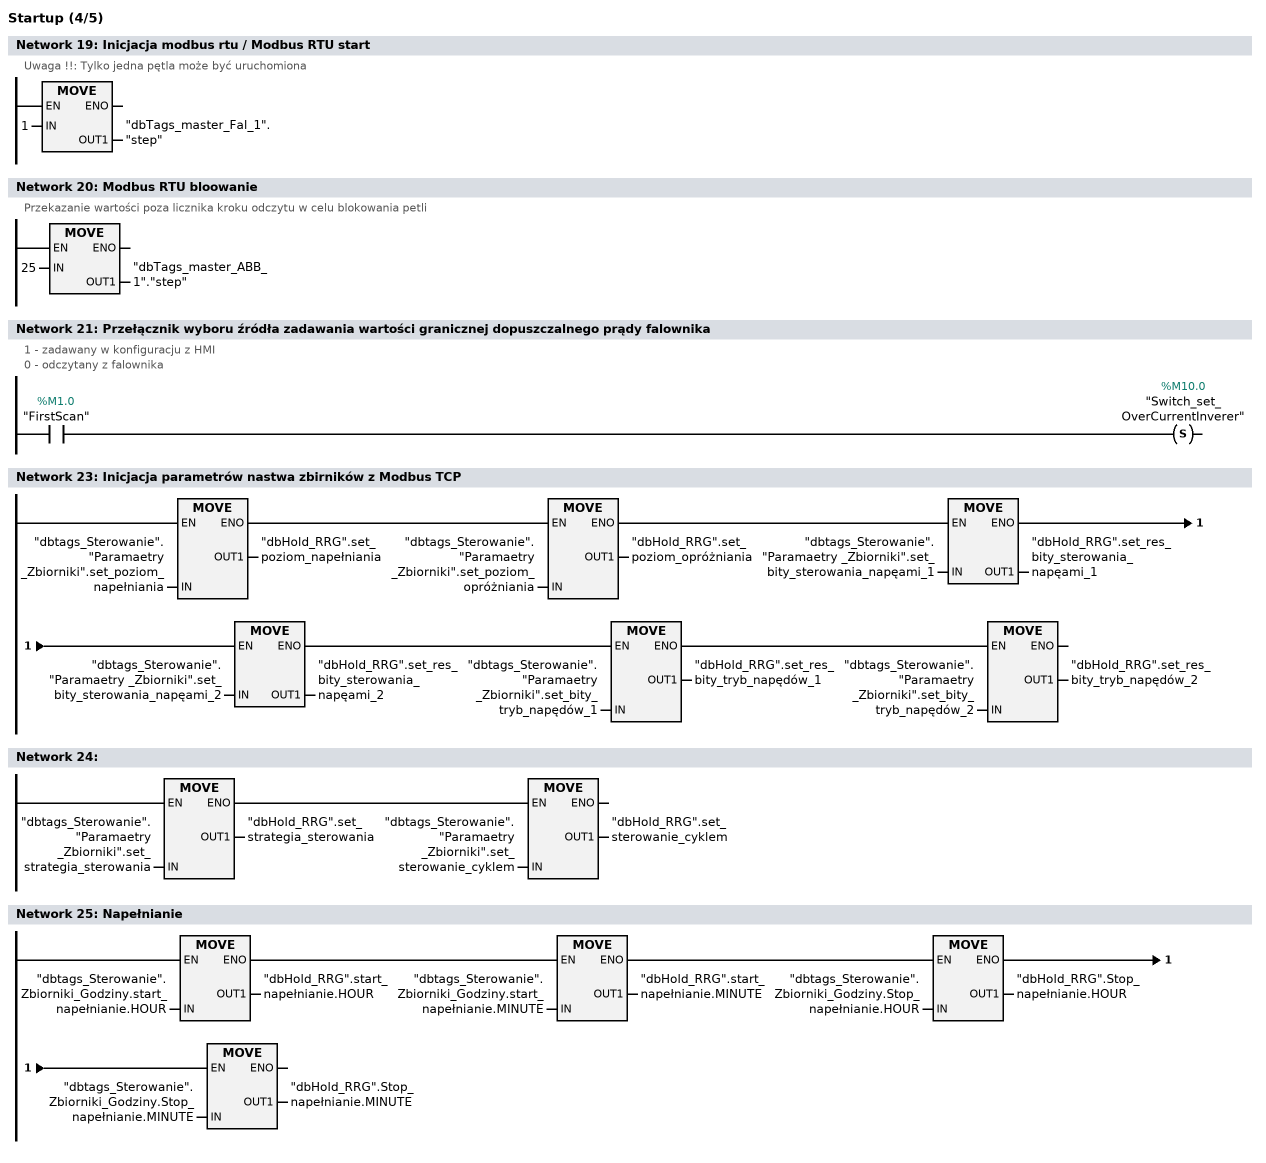
   RUNG wire#powerrail
      { S7_GenerateENO := "TRUE" } Move(in := 1, out1 => "dbTags_master_Fal_1"."step")
   END_RUNG
   // the same network as SCL:
   "dbTags_master_Fal_1"."step" := 1;
END_REGION

REGION Network 20: Modbus RTU bloowanie
   // Przekazanie wartości poza licznika kroku odczytu w celu blokowania petli
   RUNG wire#powerrail
      { S7_GenerateENO := "TRUE" } Move(in := 25, out1 => "dbTags_master_ABB_1"."step")
   END_RUNG
   // the same network as SCL:
   "dbTags_master_ABB_1"."step" := 25;
END_REGION

REGION Network 21: Przełącznik wyboru źródła zadawania wartości granicznej dopuszczalnego prądy falownika
   // 1 - zadawany w konfiguracju z HMI
   // 0 - odczytany z falownika
   RUNG wire#powerrail
      Contact( "FirstScan" )
      S_Coil( "Switch_set_OverCurrentInverer" )
   END_RUNG
   // the same network as SCL:
   IF "FirstScan" THEN "Switch_set_OverCurrentInverer" := TRUE; END_IF;
END_REGION

REGION Network 22 (SCL): Ustawienie Setpoint SV do regulatora
   // Wartość ciśnienia zadanego zależna od wybranej strategii
   CASE "dbHoldRegSlave_to_MT101".instSygSter_1 OF
     1:
       "dbdane".Setpoint_SV := "dbtags_Sterowanie".SetupControlPompownia.set_barDN500_B5 ;
     2:
       "dbdane".Setpoint_SV := "dbtags_Sterowanie".SetupControlPompownia.set_barDN225_B6;
     3:
       "dbdane".Setpoint_SV := "dbdane".Setpoint_bar_automat ;

     ELSE
       "dbdane".Setpoint_SV := 0.0;
       ;
   END_CASE;
END_REGION

REGION Network 23: Inicjacja parametrów nastwa zbirników z Modbus TCP
   RUNG wire#powerrail
      Move(in := "dbtags_Sterowanie"."Paramaetry _Zbiorniki".set_poziom_napełniania, out1 => "dbHold_RRG".set_poziom_napełniania)
      Move(in := "dbtags_Sterowanie"."Paramaetry _Zbiorniki".set_poziom_opróżniania, out1 => "dbHold_RRG".set_poziom_opróżniania)
      Move(in := "dbtags_Sterowanie"."Paramaetry _Zbiorniki".set_bity_sterowania_napęami_1, out1 => "dbHold_RRG".set_res_bity_sterowania_napęami_1)
      Move(in := "dbtags_Sterowanie"."Paramaetry _Zbiorniki".set_bity_sterowania_napęami_2, out1 => "dbHold_RRG".set_res_bity_sterowania_napęami_2)
      Move(in := "dbtags_Sterowanie"."Paramaetry _Zbiorniki".set_bity_tryb_napędów_1, out1 => "dbHold_RRG".set_res_bity_tryb_napędów_1)
      Move(in := "dbtags_Sterowanie"."Paramaetry _Zbiorniki".set_bity_tryb_napędów_2, out1 => "dbHold_RRG".set_res_bity_tryb_napędów_2)
   END_RUNG
   // the same network as SCL:
   "dbHold_RRG".set_poziom_napełniania := "dbtags_Sterowanie"."Paramaetry _Zbiorniki".set_poziom_napełniania;
   "dbHold_RRG".set_poziom_opróżniania := "dbtags_Sterowanie"."Paramaetry _Zbiorniki".set_poziom_opróżniania;
   "dbHold_RRG".set_res_bity_sterowania_napęami_1 := "dbtags_Sterowanie"."Paramaetry _Zbiorniki".set_bity_sterowania_napęami_1;
   "dbHold_RRG".set_res_bity_sterowania_napęami_2 := "dbtags_Sterowanie"."Paramaetry _Zbiorniki".set_bity_sterowania_napęami_2;
   "dbHold_RRG".set_res_bity_tryb_napędów_1 := "dbtags_Sterowanie"."Paramaetry _Zbiorniki".set_bity_tryb_napędów_1;
   "dbHold_RRG".set_res_bity_tryb_napędów_2 := "dbtags_Sterowanie"."Paramaetry _Zbiorniki".set_bity_tryb_napędów_2;
END_REGION

REGION Network 24
   RUNG wire#powerrail
      Move(in := "dbtags_Sterowanie"."Paramaetry _Zbiorniki".set_strategia_sterowania, out1 => "dbHold_RRG".set_strategia_sterowania)
      Move(in := "dbtags_Sterowanie"."Paramaetry _Zbiorniki".set_sterowanie_cyklem, out1 => "dbHold_RRG".set_sterowanie_cyklem)
   END_RUNG
   // the same network as SCL:
   "dbHold_RRG".set_strategia_sterowania := "dbtags_Sterowanie"."Paramaetry _Zbiorniki".set_strategia_sterowania;
   "dbHold_RRG".set_sterowanie_cyklem := "dbtags_Sterowanie"."Paramaetry _Zbiorniki".set_sterowanie_cyklem;
END_REGION

REGION Network 25: Napełnianie
   RUNG wire#powerrail
      Move(in := "dbtags_Sterowanie".Zbiorniki_Godziny.start_napełnianie.HOUR, out1 => "dbHold_RRG".start_napełnianie.HOUR)
      Move(in := "dbtags_Sterowanie".Zbiorniki_Godziny.start_napełnianie.MINUTE, out1 => "dbHold_RRG".start_napełnianie.MINUTE)
      Move(in := "dbtags_Sterowanie".Zbiorniki_Godziny.Stop_napełnianie.HOUR, out1 => "dbHold_RRG".Stop_napełnianie.HOUR)
      Move(in := "dbtags_Sterowanie".Zbiorniki_Godziny.Stop_napełnianie.MINUTE, out1 => "dbHold_RRG".Stop_napełnianie.MINUTE)
   END_RUNG
   // the same network as SCL:
   "dbHold_RRG".start_napełnianie.HOUR := "dbtags_Sterowanie".Zbiorniki_Godziny.start_napełnianie.HOUR;
   "dbHold_RRG".start_napełnianie.MINUTE := "dbtags_Sterowanie".Zbiorniki_Godziny.start_napełnianie.MINUTE;
   "dbHold_RRG".Stop_napełnianie.HOUR := "dbtags_Sterowanie".Zbiorniki_Godziny.Stop_napełnianie.HOUR;
   "dbHold_RRG".Stop_napełnianie.MINUTE := "dbtags_Sterowanie".Zbiorniki_Godziny.Stop_napełnianie.MINUTE;
END_REGION

REGION Network 26: Przetłaczanie
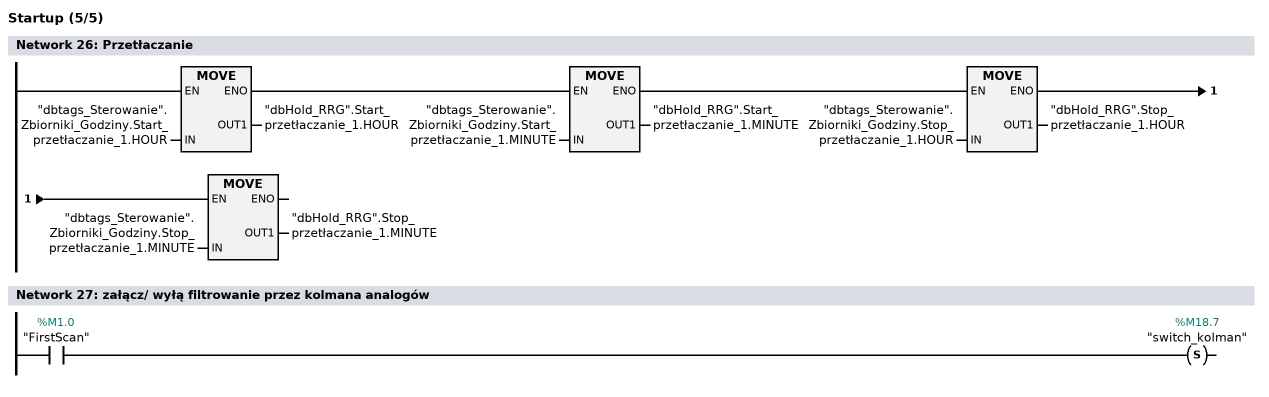
   RUNG wire#powerrail
      Move(in := "dbtags_Sterowanie".Zbiorniki_Godziny.Start_przetłaczanie_1.HOUR, out1 => "dbHold_RRG".Start_przetłaczanie_1.HOUR)
      Move(in := "dbtags_Sterowanie".Zbiorniki_Godziny.Start_przetłaczanie_1.MINUTE, out1 => "dbHold_RRG".Start_przetłaczanie_1.MINUTE)
      Move(in := "dbtags_Sterowanie".Zbiorniki_Godziny.Stop_przetłaczanie_1.HOUR, out1 => "dbHold_RRG".Stop_przetłaczanie_1.HOUR)
      Move(in := "dbtags_Sterowanie".Zbiorniki_Godziny.Stop_przetłaczanie_1.MINUTE, out1 => "dbHold_RRG".Stop_przetłaczanie_1.MINUTE)
   END_RUNG
   // the same network as SCL:
   "dbHold_RRG".Start_przetłaczanie_1.HOUR := "dbtags_Sterowanie".Zbiorniki_Godziny.Start_przetłaczanie_1.HOUR;
   "dbHold_RRG".Start_przetłaczanie_1.MINUTE := "dbtags_Sterowanie".Zbiorniki_Godziny.Start_przetłaczanie_1.MINUTE;
   "dbHold_RRG".Stop_przetłaczanie_1.HOUR := "dbtags_Sterowanie".Zbiorniki_Godziny.Stop_przetłaczanie_1.HOUR;
   "dbHold_RRG".Stop_przetłaczanie_1.MINUTE := "dbtags_Sterowanie".Zbiorniki_Godziny.Stop_przetłaczanie_1.MINUTE;
END_REGION

REGION Network 27: załącz/ wyłą filtrowanie przez kolmana analogów
   RUNG wire#powerrail
      Contact( "FirstScan" )
      S_Coil( "switch_kolman" )
   END_RUNG
   // the same network as SCL:
   IF "FirstScan" THEN "switch_kolman" := TRUE; END_IF;
END_REGION
END_ORGANIZATION_BLOCK

FUNCTION_BLOCK "00_S_WatchDog PLC - WinCC"   // FB13, LAD
TITLE = WatchDog PLC - WinCC
{ S7_Optimized_Access := 'TRUE' }
AUTHOR : rtecmer
VERSION : 0.1
// Kontrola komunikacji PLC z WinCC SCADA . Zerwanie komunikacji przekazywane do WinCC SCADA i PLC Master S7-300 (RS3)
// stored: AutoNumber true, IsIECCheckEnabled false, IsRetainMemResEnabled false, MemoryReserve 500, SetENOAutomatically false, UDAEnableTagReadback false
   VAR_TEMP   // added for the SCL form of the ladder/FBD networks
      _w1 : Bool;
      _w2 : Bool;
   END_VAR
BEGIN

REGION Network 1: WatchDog WinCC - PLC
   // Konfiguracja WinCC Flexible - ustawiony Area Point (Coordination) na DB29 DBW12
   // WinCC wpisuje z częstotliwością 0,9s na zmianę wartości 1 i 5.
   // PLC  kontroluje tę zmianę poprzez Timer TON z histerezą 10s. Jeśli nastąpi przerwanie komunikacji
   // zasygnalizuje to jeden z dwóch TON ustawiając możliwość inkrementacji zmiennej pomocniczej w instancji "Dane_ComunicationControlHMI".tempWatchDog_WinCC i ustawi bitu alarmu braku komunikacji z WinCC  
   // Po powrocie komunikacji zmienna "Dane_ComunicationControlHMI".tempWatchDog_WinCC jest zerowana.
   // Wartośc zmiennej  "Dane_ComunicationControlHMI".tempWatchDog_WinCC jest pobierana przez scipt VB WinCC jeśli jest 0 to comunikacja OK jeśli natomiast  > 0 to script VB inkrementuje wewnętrzną zmienną i ustawia alarm w WinCC.
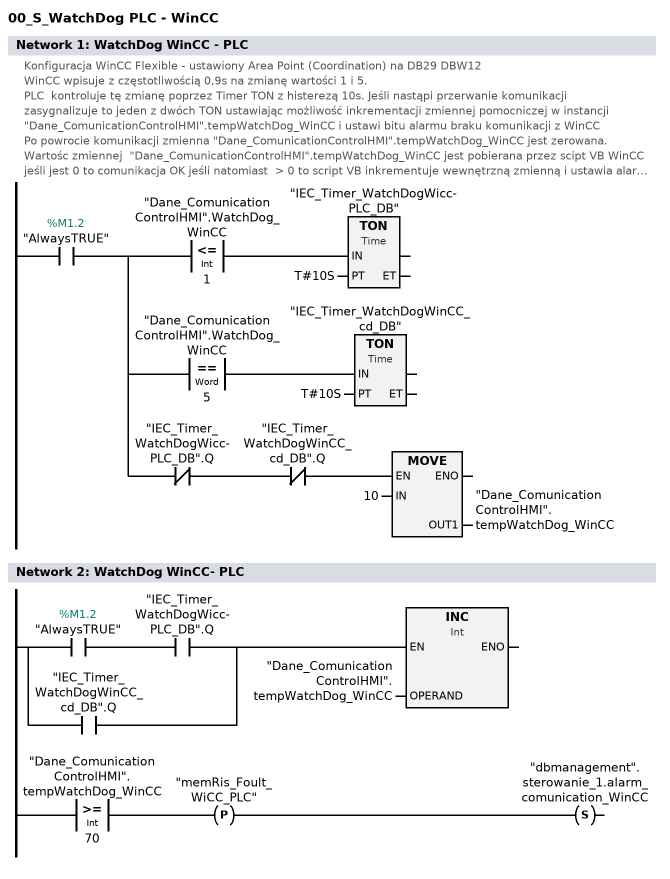
   RUNG wire#powerrail
      Contact( "AlwaysTRUE" )
      wire#w1
      { S7_Templates := "SrcType := Int" } LE_Contact(in1 := "Dane_ComunicationControlHMI".WatchDog_WinCC, in2 := 1)
      { S7_Templates := "time_type := Time" } "IEC_Timer_WatchDogWicc-PLC_DB".TON(pt := T#10S, et =>)
   END_RUNG
   RUNG wire#w1
      { S7_Templates := "SrcType := Word" } EQ_Contact(in1 := "Dane_ComunicationControlHMI".WatchDog_WinCC, in2 := 5)
      { S7_Templates := "time_type := Time" } "IEC_Timer_WatchDogWinCC_cd_DB".TON(pt := T#10S, et =>)
   END_RUNG
   RUNG wire#w1
      I_Contact( "IEC_Timer_WatchDogWicc-PLC_DB".Q )
      I_Contact( "IEC_Timer_WatchDogWinCC_cd_DB".Q )
      Move(in := 10, out1 => "Dane_ComunicationControlHMI".tempWatchDog_WinCC)
   END_RUNG
   // the same network as SCL:
   "IEC_Timer_WatchDogWicc-PLC_DB".TON(IN := "AlwaysTRUE" AND ("Dane_ComunicationControlHMI".WatchDog_WinCC <= 1),
                           PT := T#10S);
   "IEC_Timer_WatchDogWinCC_cd_DB".TON(IN := "AlwaysTRUE" AND ("Dane_ComunicationControlHMI".WatchDog_WinCC = 5),
                           PT := T#10S);
   IF "AlwaysTRUE" AND NOT "IEC_Timer_WatchDogWicc-PLC_DB".Q AND NOT "IEC_Timer_WatchDogWinCC_cd_DB".Q THEN
       "Dane_ComunicationControlHMI".tempWatchDog_WinCC := 10;
   END_IF;
END_REGION

